Yaskawa INFORM job: DEMO_ROOF_SIDE_0625_3PAINT_44.JBI

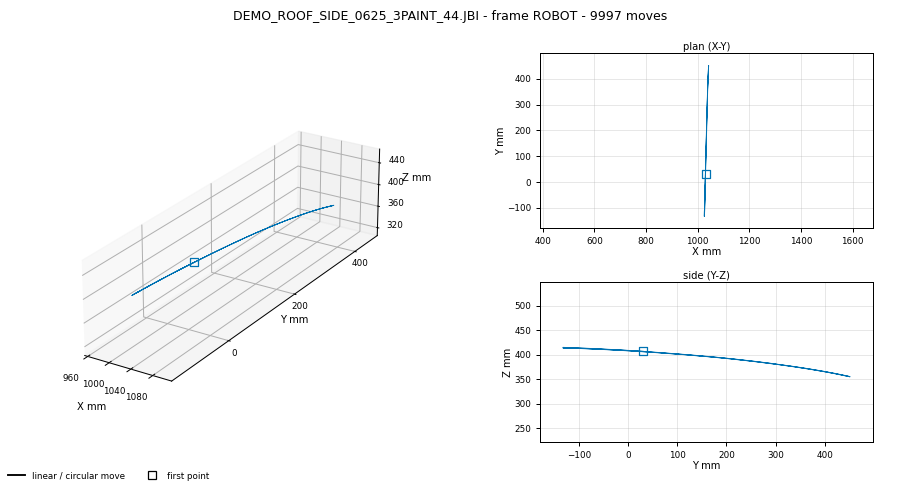
[picture p0: tool path of DEMO_ROOF_SIDE_0625_3PAINT_44.JBI in frame ROBOT, 9997 of 9997 moves have a stored position in this frame; points joined in program order, loops and branches not executed]
/JOB
//NAME DEMO_ROOF_SIDE_0625_3PAINT44
//POS
///NPOS 9997,0,0,0,0,0
///TOOL 0
///USER 0
///POSTYPE ROBOT
///RECTAN
///RCONF 1,0,0,0,0,0,0,0,0,0,0,0,0,0,0,0,0,0,0,0,0,0,0,0
C00000=1030.820,31.056,407.036,168.328,43.418,158.095
C00001=1030.814,30.807,407.052,168.325,43.419,158.095
C00002=1030.807,30.558,407.068,168.324,43.421,158.095
C00003=1030.801,30.309,407.084,168.321,43.422,158.095
C00004=1030.795,30.059,407.101,168.319,43.423,158.096
C00005=1030.788,29.809,407.116,168.316,43.425,158.096
C00006=1030.782,29.560,407.132,168.314,43.426,158.096
C00007=1030.776,29.310,407.148,168.312,43.427,158.096
C00008=1030.770,29.061,407.164,168.309,43.429,158.096
C00009=1030.764,28.812,407.180,168.306,43.431,158.096
C00010=1030.758,28.562,407.197,168.305,43.432,158.096
C00011=1030.750,28.276,407.215,168.302,43.433,158.096
C00012=1030.744,27.990,407.233,168.299,43.435,158.096
C00013=1030.737,27.704,407.251,168.297,43.437,158.096
C00014=1030.728,27.418,407.269,168.294,43.438,158.096
C00015=1030.722,27.169,407.286,168.291,43.440,158.096
C00016=1030.716,26.919,407.301,168.289,43.442,158.097
C00017=1030.710,26.670,407.317,168.287,43.443,158.097
C00018=1030.703,26.421,407.333,168.284,43.445,158.097
C00019=1030.697,26.171,407.349,168.281,43.446,158.097
C00020=1030.692,25.921,407.364,168.280,43.448,158.097
C00021=1030.685,25.672,407.380,168.277,43.449,158.097
C00022=1030.678,25.422,407.396,168.274,43.451,158.097
C00023=1030.672,25.173,407.412,168.272,43.452,158.097
C00024=1030.665,24.923,407.427,168.270,43.454,158.097
C00025=1030.660,24.674,407.444,168.267,43.456,158.097
C00026=1030.653,24.425,407.459,168.265,43.457,158.097
C00027=1030.647,24.175,407.475,168.263,43.459,158.098
C00028=1030.641,23.926,407.490,168.260,43.460,158.098
C00029=1030.635,23.677,407.507,168.257,43.462,158.098
C00030=1030.628,23.427,407.522,168.255,43.463,158.098
C00031=1030.622,23.178,407.538,168.253,43.464,158.098
C00032=1030.616,22.929,407.554,168.250,43.466,158.098
C00033=1030.610,22.679,407.569,168.248,43.467,158.098
C00034=1030.603,22.430,407.585,168.245,43.469,158.098
C00035=1030.597,22.181,407.600,168.243,43.470,158.098
C00036=1030.591,21.931,407.616,168.241,43.471,158.098
C00037=1030.584,21.682,407.632,168.238,43.473,158.098
C00038=1030.579,21.432,407.647,168.236,43.474,158.098
C00039=1030.572,21.183,407.663,168.234,43.476,158.098
C00040=1030.566,20.933,407.679,168.231,43.477,158.098
C00041=1030.560,20.684,407.694,168.228,43.479,158.099
C00042=1030.554,20.434,407.710,168.227,43.480,158.099
C00043=1030.547,20.185,407.725,168.224,43.482,158.099
C00044=1030.540,19.936,407.741,168.221,43.483,158.099
C00045=1030.535,19.686,407.756,168.220,43.485,158.099
C00046=1030.528,19.437,407.772,168.217,43.487,158.099
C00047=1030.523,19.187,407.788,168.214,43.488,158.099
C00048=1030.516,18.938,407.803,168.212,43.490,158.099
C00049=1030.509,18.688,407.818,168.210,43.491,158.099
C00050=1030.503,18.439,407.834,168.207,43.493,158.099
C00051=1030.497,18.189,407.849,168.204,43.494,158.099
C00052=1030.490,17.940,407.865,168.203,43.496,158.100
C00053=1030.484,17.690,407.880,168.200,43.498,158.100
C00054=1030.478,17.441,407.896,168.197,43.499,158.100
C00055=1030.472,17.191,407.911,168.195,43.500,158.100
C00056=1030.465,16.942,407.926,168.193,43.502,158.100
C00057=1030.459,16.692,407.942,168.190,43.504,158.100
C00058=1030.453,16.442,407.957,168.188,43.505,158.100
C00059=1030.446,16.193,407.973,168.186,43.506,158.100
C00060=1030.440,15.944,407.988,168.183,43.508,158.100
C00061=1030.434,15.694,408.004,168.180,43.509,158.100
C00062=1030.428,15.445,408.019,168.178,43.511,158.100
C00063=1030.421,15.195,408.034,168.176,43.512,158.100
C00064=1030.416,14.947,408.050,168.173,43.514,158.101
C00065=1030.409,14.697,408.065,168.171,43.515,158.101
C00066=1030.403,14.447,408.080,168.169,43.517,158.101
C00067=1030.396,14.198,408.096,168.166,43.518,158.101
C00068=1030.391,13.948,408.111,168.164,43.520,158.101
C00069=1030.384,13.699,408.126,168.161,43.521,158.101
C00070=1030.378,13.449,408.142,168.159,43.523,158.101
C00071=1030.371,13.200,408.157,168.156,43.525,158.101
C00072=1030.365,12.950,408.172,168.154,43.526,158.101
C00073=1030.359,12.701,408.187,168.151,43.528,158.101
C00074=1030.352,12.451,408.202,168.149,43.530,158.101
C00075=1030.345,12.166,408.219,168.146,43.531,158.101
C00076=1030.338,11.882,408.236,168.143,43.533,158.102
C00077=1030.330,11.597,408.253,168.141,43.535,158.102
C00078=1030.323,11.312,408.271,168.137,43.537,158.102
C00079=1030.317,11.063,408.285,168.136,43.538,158.102
C00080=1030.310,10.813,408.300,168.133,43.540,158.102
C00081=1030.304,10.563,408.315,168.130,43.541,158.102
C00082=1030.298,10.314,408.330,168.127,43.543,158.102
C00083=1030.291,10.065,408.346,168.126,43.544,158.102
C00084=1030.285,9.816,408.361,168.123,43.546,158.102
C00085=1030.279,9.566,408.376,168.120,43.548,158.103
C00086=1030.272,9.317,408.390,168.117,43.549,158.102
C00087=1030.266,9.067,408.405,168.116,43.551,158.103
C00088=1030.260,8.817,408.420,168.113,43.553,158.103
C00089=1030.253,8.568,408.435,168.110,43.554,158.103
C00090=1030.247,8.319,408.450,168.108,43.556,158.103
C00091=1030.241,8.069,408.465,168.105,43.558,158.103
C00092=1030.234,7.820,408.480,168.103,43.559,158.103
C00093=1030.228,7.570,408.495,168.101,43.561,158.103
C00094=1030.222,7.321,408.510,168.098,43.562,158.103
C00095=1030.215,7.071,408.525,168.095,43.564,158.103
C00096=1030.209,6.822,408.540,168.094,43.566,158.104
C00097=1030.203,6.572,408.555,168.091,43.567,158.104
C00098=1030.197,6.323,408.570,168.088,43.569,158.104
C00099=1030.190,6.073,408.585,168.085,43.570,158.104
C00100=1030.184,5.824,408.599,168.084,43.572,158.104
C00101=1030.178,5.574,408.614,168.081,43.573,158.104
C00102=1030.172,5.325,408.629,168.078,43.575,158.104
C00103=1030.165,5.075,408.644,168.076,43.576,158.104
C00104=1030.159,4.825,408.659,168.074,43.577,158.104
C00105=1030.153,4.576,408.674,168.071,43.579,158.104
C00106=1030.147,4.327,408.689,168.068,43.581,158.104
C00107=1030.140,4.077,408.704,168.066,43.582,158.104
C00108=1030.134,3.827,408.719,168.063,43.584,158.104
C00109=1030.128,3.579,408.733,168.061,43.585,158.104
C00110=1030.122,3.329,408.748,168.059,43.587,158.105
C00111=1030.115,3.079,408.763,168.056,43.588,158.105
C00112=1030.110,2.830,408.778,168.053,43.590,158.105
C00113=1030.103,2.581,408.793,168.051,43.592,158.105
C00114=1030.097,2.331,408.807,168.049,43.593,158.105
C00115=1030.090,2.081,408.822,168.046,43.595,158.105
C00116=1030.085,1.832,408.836,168.043,43.596,158.105
C00117=1030.079,1.582,408.851,168.042,43.598,158.105
C00118=1030.072,1.332,408.866,168.039,43.599,158.105
C00119=1030.066,1.083,408.881,168.036,43.601,158.105
C00120=1030.060,0.834,408.896,168.033,43.602,158.105
C00121=1030.054,0.584,408.911,168.032,43.604,158.105
C00122=1030.048,0.335,408.925,168.029,43.605,158.105
C00123=1030.042,0.086,408.940,168.026,43.607,158.106
C00124=1030.035,-0.165,408.954,168.023,43.608,158.106
C00125=1030.030,-0.414,408.969,168.021,43.610,158.106
C00126=1030.023,-0.663,408.983,168.019,43.612,158.106
C00127=1030.016,-0.913,408.998,168.016,43.613,158.106
C00128=1030.010,-1.162,409.013,168.014,43.615,158.106
C00129=1030.004,-1.411,409.028,168.011,43.616,158.106
C00130=1029.999,-1.661,409.042,168.009,43.618,158.106
C00131=1029.992,-1.911,409.057,168.006,43.619,158.106
C00132=1029.986,-2.160,409.072,168.004,43.621,158.106
C00133=1029.980,-2.409,409.086,168.001,43.622,158.106
C00134=1029.974,-2.659,409.101,167.999,43.624,158.106
C00135=1029.968,-2.908,409.115,167.996,43.625,158.106
C00136=1029.962,-3.158,409.130,167.994,43.627,158.107
C00137=1029.955,-3.408,409.145,167.991,43.628,158.107
C00138=1029.950,-3.657,409.159,167.989,43.630,158.107
C00139=1029.942,-3.940,409.176,167.985,43.631,158.107
C00140=1029.935,-4.223,409.191,167.983,43.633,158.107
C00141=1029.928,-4.505,409.208,167.980,43.635,158.107
C00142=1029.921,-4.789,409.225,167.978,43.637,158.107
C00143=1029.915,-5.038,409.238,167.975,43.639,158.107
C00144=1029.908,-5.288,409.253,167.972,43.641,158.107
C00145=1029.902,-5.537,409.267,167.969,43.642,158.107
C00146=1029.896,-5.787,409.281,167.967,43.644,158.107
C00147=1029.889,-6.036,409.296,167.964,43.646,158.107
C00148=1029.883,-6.286,409.309,167.962,43.647,158.108
C00149=1029.877,-6.535,409.324,167.960,43.649,158.108
C00150=1029.871,-6.784,409.339,167.957,43.650,158.108
C00151=1029.864,-7.034,409.352,167.954,43.652,158.108
C00152=1029.858,-7.284,409.367,167.952,43.654,158.108
C00153=1029.851,-7.533,409.381,167.949,43.655,158.108
C00154=1029.845,-7.783,409.396,167.946,43.657,158.108
C00155=1029.840,-8.032,409.409,167.945,43.658,158.108
C00156=1029.832,-8.282,409.424,167.942,43.660,158.108
C00157=1029.827,-8.531,409.438,167.939,43.661,158.108
C00158=1029.820,-8.781,409.452,167.936,43.663,158.108
C00159=1029.814,-9.030,409.466,167.934,43.665,158.109
C00160=1029.808,-9.280,409.481,167.931,43.666,158.109
C00161=1029.801,-9.530,409.494,167.928,43.668,158.109
C00162=1029.795,-9.779,409.509,167.927,43.670,158.109
C00163=1029.789,-10.029,409.523,167.924,43.671,158.109
C00164=1029.783,-10.278,409.537,167.921,43.673,158.109
C00165=1029.776,-10.528,409.551,167.919,43.675,158.109
C00166=1029.770,-10.777,409.565,167.916,43.676,158.109
C00167=1029.764,-11.027,409.580,167.913,43.678,158.109
C00168=1029.758,-11.276,409.593,167.911,43.680,158.109
C00169=1029.752,-11.526,409.608,167.909,43.681,158.109
C00170=1029.745,-11.775,409.621,167.906,43.683,158.109
C00171=1029.740,-12.025,409.635,167.903,43.684,158.109
C00172=1029.733,-12.274,409.649,167.901,43.686,158.110
C00173=1029.727,-12.524,409.663,167.898,43.688,158.110
C00174=1029.721,-12.773,409.678,167.895,43.689,158.110
C00175=1029.715,-13.023,409.691,167.893,43.691,158.110
C00176=1029.709,-13.273,409.706,167.891,43.693,158.110
C00177=1029.702,-13.521,409.720,167.888,43.694,158.110
C00178=1029.696,-13.772,409.734,167.885,43.696,158.110
C00179=1029.690,-14.021,409.747,167.883,43.697,158.110
C00180=1029.684,-14.270,409.762,167.880,43.699,158.110
C00181=1029.678,-14.520,409.776,167.877,43.701,158.110
C00182=1029.672,-14.770,409.789,167.875,43.702,158.110
C00183=1029.666,-15.020,409.803,167.873,43.704,158.110
C00184=1029.659,-15.268,409.817,167.870,43.705,158.110
C00185=1029.653,-15.519,409.832,167.867,43.707,158.111
C00186=1029.647,-15.768,409.845,167.865,43.709,158.111
C00187=1029.640,-16.018,409.859,167.862,43.710,158.111
C00188=1029.634,-16.267,409.873,167.859,43.712,158.111
C00189=1029.628,-16.516,409.886,167.857,43.714,158.111
C00190=1029.621,-16.766,409.900,167.854,43.716,158.111
C00191=1029.616,-17.016,409.914,167.851,43.717,158.111
C00192=1029.609,-17.266,409.928,167.849,43.719,158.111
C00193=1029.603,-17.515,409.941,167.847,43.720,158.111
C00194=1029.597,-17.764,409.955,167.844,43.722,158.111
C00195=1029.590,-18.014,409.969,167.842,43.723,158.111
C00196=1029.584,-18.263,409.982,167.839,43.725,158.112
C00197=1029.578,-18.513,409.997,167.836,43.727,158.112
C00198=1029.572,-18.763,410.010,167.834,43.729,158.112
C00199=1029.565,-19.012,410.023,167.831,43.730,158.112
C00200=1029.559,-19.262,410.037,167.828,43.732,158.112
C00201=1029.553,-19.511,410.051,167.826,43.734,158.112
C00202=1029.547,-19.761,410.064,167.823,43.736,158.112
C00203=1029.540,-20.042,410.080,167.820,43.738,158.112
C00204=1029.533,-20.323,410.095,167.817,43.739,158.112
C00205=1029.525,-20.605,410.110,167.814,43.741,158.112
C00206=1029.518,-20.886,410.126,167.811,43.743,158.112
C00207=1029.512,-21.135,410.139,167.809,43.745,158.113
C00208=1029.506,-21.385,410.153,167.806,43.747,158.113
C00209=1029.500,-21.635,410.167,167.803,43.748,158.113
C00210=1029.493,-21.884,410.180,167.800,43.750,158.113
C00211=1029.487,-22.134,410.193,167.798,43.752,158.113
C00212=1029.482,-22.383,410.207,167.795,43.754,158.113
C00213=1029.475,-22.633,410.221,167.793,43.755,158.113
C00214=1029.469,-22.882,410.234,167.791,43.757,158.113
C00215=1029.463,-23.132,410.248,167.788,43.759,158.113
C00216=1029.456,-23.382,410.261,167.785,43.760,158.113
C00217=1029.450,-23.631,410.275,167.783,43.762,158.113
C00218=1029.444,-23.880,410.288,167.780,43.764,158.113
C00219=1029.438,-24.130,410.302,167.777,43.765,158.113
C00220=1029.432,-24.380,410.316,167.775,43.767,158.114
C00221=1029.425,-24.629,410.329,167.772,43.769,158.114
C00222=1029.419,-24.878,410.342,167.769,43.770,158.114
C00223=1029.414,-25.128,410.356,167.766,43.772,158.114
C00224=1029.407,-25.378,410.370,167.764,43.774,158.114
C00225=1029.401,-25.628,410.382,167.761,43.775,158.114
C00226=1029.395,-25.877,410.395,167.758,43.777,158.114
C00227=1029.389,-26.127,410.409,167.756,43.779,158.114
C00228=1029.383,-26.376,410.423,167.754,43.780,158.114
C00229=1029.376,-26.626,410.436,167.751,43.782,158.114
C00230=1029.370,-26.875,410.449,167.749,43.783,158.114
C00231=1029.365,-27.125,410.463,167.746,43.785,158.114
C00232=1029.359,-27.375,410.476,167.743,43.787,158.115
C00233=1029.352,-27.625,410.489,167.741,43.788,158.115
C00234=1029.346,-27.874,410.503,167.738,43.790,158.115
C00235=1029.339,-28.123,410.516,167.735,43.792,158.115
C00236=1029.334,-28.373,410.529,167.732,43.793,158.115
C00237=1029.327,-28.622,410.542,167.730,43.795,158.115
C00238=1029.321,-28.872,410.555,167.727,43.797,158.115
C00239=1029.314,-29.122,410.569,167.725,43.799,158.115
C00240=1029.308,-29.371,410.581,167.722,43.801,158.115
C00241=1029.302,-29.621,410.595,167.719,43.802,158.115
C00242=1029.296,-29.870,410.608,167.716,43.804,158.115
C00243=1029.289,-30.121,410.621,167.714,43.806,158.116
C00244=1029.283,-30.370,410.634,167.711,43.808,158.116
C00245=1029.277,-30.619,410.647,167.709,43.810,158.116
C00246=1029.271,-30.869,410.660,167.706,43.811,158.116
C00247=1029.265,-31.118,410.673,167.703,43.813,158.116
C00248=1029.259,-31.367,410.686,167.701,43.815,158.116
C00249=1029.253,-31.617,410.699,167.698,43.817,158.116
C00250=1029.246,-31.867,410.713,167.695,43.818,158.116
C00251=1029.240,-32.117,410.726,167.692,43.820,158.116
C00252=1029.234,-32.366,410.738,167.690,43.822,158.116
C00253=1029.228,-32.616,410.752,167.687,43.824,158.116
C00254=1029.222,-32.866,410.764,167.685,43.826,158.117
C00255=1029.216,-33.115,410.777,167.682,43.827,158.117
C00256=1029.209,-33.364,410.791,167.679,43.829,158.117
C00257=1029.203,-33.614,410.803,167.676,43.831,158.117
C00258=1029.196,-33.864,410.816,167.674,43.833,158.117
C00259=1029.190,-34.114,410.829,167.671,43.834,158.117
C00260=1029.184,-34.363,410.842,167.668,43.836,158.117
C00261=1029.178,-34.613,410.855,167.666,43.838,158.117
C00262=1029.172,-34.862,410.868,167.663,43.840,158.117
C00263=1029.166,-35.112,410.881,167.660,43.841,158.117
C00264=1029.159,-35.361,410.894,167.658,43.843,158.117
C00265=1029.154,-35.611,410.906,167.655,43.845,158.117
C00266=1029.147,-35.860,410.920,167.652,43.846,158.118
C00267=1029.141,-36.141,410.934,167.649,43.849,158.118
C00268=1029.134,-36.421,410.948,167.646,43.850,158.118
C00269=1029.127,-36.702,410.963,167.643,43.852,158.118
C00270=1029.120,-36.982,410.977,167.640,43.854,158.118
C00271=1029.114,-37.232,410.990,167.637,43.856,158.118
C00272=1029.108,-37.481,411.003,167.634,43.858,158.118
C00273=1029.102,-37.731,411.016,167.632,43.859,158.118
C00274=1029.095,-37.980,411.029,167.629,43.861,158.118
C00275=1029.090,-38.230,411.042,167.626,43.863,158.118
C00276=1029.084,-38.480,411.054,167.624,43.864,158.118
C00277=1029.077,-38.729,411.067,167.621,43.866,158.118
C00278=1029.072,-38.979,411.080,167.618,43.868,158.118
C00279=1029.065,-39.228,411.093,167.616,43.870,158.119
C00280=1029.059,-39.478,411.105,167.613,43.871,158.119
C00281=1029.053,-39.728,411.118,167.610,43.873,158.119
C00282=1029.047,-39.978,411.130,167.608,43.875,158.119
C00283=1029.040,-40.227,411.143,167.605,43.877,158.119
C00284=1029.034,-40.476,411.155,167.602,43.879,158.119
C00285=1029.028,-40.726,411.168,167.600,43.881,158.119
C00286=1029.022,-40.976,411.181,167.596,43.882,158.119
C00287=1029.015,-41.225,411.193,167.593,43.884,158.119
C00288=1029.009,-41.475,411.206,167.591,43.886,158.119
C00289=1029.003,-41.725,411.218,167.588,43.888,158.119
C00290=1028.996,-41.974,411.231,167.585,43.890,158.120
C00291=1028.991,-42.224,411.244,167.583,43.892,158.120
C00292=1028.985,-42.474,411.256,167.580,43.894,158.120
C00293=1028.978,-42.723,411.268,167.578,43.896,158.120
C00294=1028.972,-42.973,411.281,167.575,43.897,158.120
C00295=1028.966,-43.222,411.294,167.572,43.899,158.120
C00296=1028.959,-43.472,411.306,167.569,43.901,158.120
C00297=1028.953,-43.722,411.318,167.567,43.903,158.120
C00298=1028.948,-43.971,411.331,167.563,43.905,158.120
C00299=1028.941,-44.221,411.343,167.561,43.907,158.120
C00300=1028.935,-44.471,411.355,167.558,43.909,158.121
C00301=1028.929,-44.720,411.368,167.555,43.910,158.120
C00302=1028.923,-44.969,411.380,167.552,43.912,158.121
C00303=1028.917,-45.219,411.393,167.550,43.914,158.121
C00304=1028.911,-45.469,411.405,167.547,43.916,158.121
C00305=1028.904,-45.719,411.417,167.545,43.917,158.121
C00306=1028.898,-45.969,411.430,167.542,43.919,158.121
C00307=1028.893,-46.218,411.442,167.539,43.921,158.121
C00308=1028.886,-46.467,411.454,167.536,43.923,158.121
C00309=1028.880,-46.717,411.467,167.534,43.924,158.121
C00310=1028.874,-46.966,411.480,167.531,43.926,158.121
C00311=1028.867,-47.216,411.492,167.528,43.928,158.121
C00312=1028.862,-47.466,411.504,167.525,43.930,158.122
C00313=1028.856,-47.715,411.517,167.522,43.932,158.122
C00314=1028.850,-47.965,411.529,167.520,43.933,158.122
C00315=1028.844,-48.215,411.541,167.517,43.935,158.122
C00316=1028.838,-48.464,411.554,167.514,43.937,158.122
C00317=1028.831,-48.714,411.566,167.512,43.939,158.122
C00318=1028.826,-48.963,411.578,167.509,43.940,158.122
C00319=1028.819,-49.213,411.590,167.506,43.942,158.122
C00320=1028.813,-49.463,411.602,167.504,43.944,158.122
C00321=1028.807,-49.713,411.615,167.501,43.946,158.122
C00322=1028.801,-49.962,411.627,167.498,43.948,158.122
C00323=1028.795,-50.211,411.639,167.494,43.950,158.122
C00324=1028.790,-50.461,411.652,167.492,43.951,158.122
C00325=1028.783,-50.711,411.664,167.489,43.953,158.123
C00326=1028.777,-50.961,411.675,167.487,43.955,158.123
C00327=1028.771,-51.211,411.687,167.484,43.957,158.123
C00328=1028.765,-51.460,411.699,167.481,43.959,158.123
C00329=1028.758,-51.709,411.711,167.479,43.961,158.123
C00330=1028.752,-51.959,411.724,167.475,43.963,158.123
C00331=1028.743,-52.314,411.740,167.472,43.966,158.123
C00332=1028.734,-52.667,411.757,167.467,43.969,158.123
C00333=1028.725,-53.021,411.774,167.464,43.972,158.124
C00334=1028.717,-53.376,411.791,167.459,43.975,158.124
C00335=1028.710,-53.625,411.803,167.457,43.977,158.124
C00336=1028.704,-53.874,411.814,167.454,43.978,158.124
C00337=1028.698,-54.124,411.825,167.451,43.980,158.124
C00338=1028.692,-54.374,411.838,167.449,43.982,158.124
C00339=1028.685,-54.624,411.850,167.445,43.984,158.124
C00340=1028.679,-54.873,411.861,167.443,43.986,158.124
C00341=1028.673,-55.123,411.873,167.440,43.988,158.124
C00342=1028.667,-55.373,411.885,167.437,43.990,158.125
C00343=1028.661,-55.622,411.897,167.435,43.992,158.125
C00344=1028.654,-55.872,411.908,167.431,43.994,158.125
C00345=1028.648,-56.121,411.920,167.428,43.996,158.125
C00346=1028.642,-56.371,411.932,167.426,43.998,158.125
C00347=1028.636,-56.621,411.943,167.423,44.000,158.125
C00348=1028.629,-56.870,411.955,167.421,44.002,158.125
C00349=1028.623,-57.120,411.967,167.417,44.004,158.125
C00350=1028.618,-57.370,411.979,167.414,44.006,158.125
C00351=1028.611,-57.619,411.991,167.412,44.008,158.125
C00352=1028.605,-57.869,412.002,167.409,44.010,158.126
C00353=1028.599,-58.118,412.014,167.406,44.012,158.126
C00354=1028.593,-58.369,412.026,167.404,44.014,158.126
C00355=1028.587,-58.618,412.037,167.400,44.016,158.126
C00356=1028.580,-58.867,412.049,167.397,44.018,158.126
C00357=1028.574,-59.117,412.060,167.395,44.019,158.126
C00358=1028.568,-59.366,412.072,167.392,44.021,158.126
C00359=1028.562,-59.617,412.084,167.390,44.023,158.126
C00360=1028.556,-59.866,412.096,167.386,44.025,158.126
C00361=1028.550,-60.116,412.107,167.383,44.027,158.126
C00362=1028.543,-60.365,412.119,167.381,44.029,158.126
C00363=1028.538,-60.615,412.130,167.378,44.031,158.127
C00364=1028.532,-60.865,412.142,167.375,44.033,158.127
C00365=1028.526,-61.114,412.153,167.372,44.035,158.127
C00366=1028.519,-61.364,412.165,167.369,44.037,158.127
C00367=1028.513,-61.614,412.176,167.367,44.039,158.127
C00368=1028.508,-61.863,412.188,167.364,44.041,158.127
C00369=1028.501,-62.113,412.199,167.361,44.043,158.127
C00370=1028.495,-62.362,412.211,167.358,44.045,158.127
C00371=1028.489,-62.613,412.222,167.355,44.047,158.127
C00372=1028.483,-62.861,412.234,167.352,44.049,158.127
C00373=1028.477,-63.112,412.246,167.350,44.051,158.128
C00374=1028.471,-63.361,412.257,167.347,44.053,158.128
C00375=1028.465,-63.611,412.269,167.344,44.055,158.128
C00376=1028.459,-63.860,412.279,167.341,44.057,158.128
C00377=1028.453,-64.110,412.291,167.338,44.059,158.128
C00378=1028.448,-64.360,412.303,167.336,44.061,158.128
C00379=1028.441,-64.609,412.315,167.333,44.063,158.128
C00380=1028.435,-64.859,412.326,167.330,44.064,158.128
C00381=1028.429,-65.109,412.337,167.327,44.067,158.128
C00382=1028.423,-65.358,412.349,167.324,44.068,158.128
C00383=1028.417,-65.608,412.360,167.322,44.070,158.129
C00384=1028.412,-65.858,412.371,167.319,44.072,158.129
C00385=1028.405,-66.107,412.383,167.316,44.074,158.129
C00386=1028.399,-66.357,412.394,167.313,44.076,158.129
C00387=1028.393,-66.570,412.404,167.311,44.077,158.129
C00388=1028.389,-66.783,412.414,167.308,44.079,158.129
C00389=1028.384,-66.997,412.423,167.306,44.081,158.129
C00390=1028.379,-67.209,412.433,167.303,44.083,158.129
C00391=1028.373,-67.423,412.443,167.301,44.084,158.129
C00392=1028.368,-67.636,412.453,167.299,44.086,158.129
C00393=1028.364,-67.849,412.462,167.296,44.087,158.129
C00394=1028.358,-68.062,412.472,167.294,44.089,158.129
C00395=1028.352,-68.344,412.484,167.290,44.091,158.129
C00396=1028.345,-68.626,412.498,167.287,44.093,158.130
C00397=1028.338,-68.908,412.510,167.284,44.096,158.130
C00398=1028.331,-69.191,412.523,167.281,44.098,158.130
C00399=1028.325,-69.440,412.534,167.278,44.100,158.130
C00400=1028.320,-69.690,412.545,167.275,44.102,158.130
C00401=1028.314,-69.940,412.557,167.272,44.104,158.130
C00402=1028.308,-70.189,412.568,167.269,44.106,158.130
C00403=1028.302,-70.439,412.579,167.266,44.107,158.130
C00404=1028.296,-70.689,412.590,167.264,44.109,158.130
C00405=1028.290,-70.938,412.601,167.261,44.111,158.130
C00406=1028.284,-71.188,412.612,167.257,44.113,158.130
C00407=1028.278,-71.437,412.624,167.255,44.115,158.130
C00408=1028.273,-71.687,412.635,167.252,44.117,158.131
C00409=1028.267,-71.937,412.646,167.250,44.119,158.131
C00410=1028.261,-72.187,412.658,167.247,44.121,158.131
C00411=1028.255,-72.436,412.668,167.243,44.123,158.131
C00412=1028.249,-72.686,412.679,167.241,44.125,158.131
C00413=1028.243,-72.936,412.691,167.238,44.127,158.131
C00414=1028.237,-73.185,412.701,167.235,44.129,158.131
C00415=1028.232,-73.435,412.713,167.233,44.131,158.131
C00416=1028.225,-73.685,412.725,167.229,44.132,158.131
C00417=1028.220,-73.934,412.736,167.226,44.134,158.131
C00418=1028.214,-74.184,412.747,167.224,44.136,158.131
C00419=1028.208,-74.433,412.757,167.221,44.138,158.131
C00420=1028.202,-74.684,412.769,167.219,44.140,158.132
C00421=1028.196,-74.933,412.780,167.215,44.143,158.132
C00422=1028.190,-75.182,412.790,167.212,44.145,158.132
C00423=1028.184,-75.433,412.800,167.210,44.147,158.132
C00424=1028.178,-75.682,412.811,167.206,44.149,158.132
C00425=1028.172,-75.932,412.822,167.204,44.151,158.132
C00426=1028.166,-76.181,412.833,167.201,44.153,158.132
C00427=1028.160,-76.432,412.844,167.198,44.155,158.132
C00428=1028.154,-76.681,412.855,167.195,44.157,158.132
C00429=1028.148,-76.930,412.865,167.192,44.159,158.132
C00430=1028.141,-77.181,412.877,167.189,44.161,158.133
C00431=1028.136,-77.430,412.888,167.187,44.163,158.133
C00432=1028.130,-77.679,412.898,167.183,44.165,158.133
C00433=1028.125,-77.930,412.909,167.181,44.167,158.133
C00434=1028.119,-78.179,412.920,167.178,44.169,158.133
C00435=1028.112,-78.429,412.930,167.175,44.171,158.133
C00436=1028.106,-78.678,412.941,167.172,44.173,158.133
C00437=1028.100,-78.928,412.952,167.169,44.175,158.133
C00438=1028.094,-79.177,412.963,167.167,44.177,158.133
C00439=1028.088,-79.428,412.973,167.163,44.179,158.133
C00440=1028.083,-79.678,412.984,167.160,44.181,158.134
C00441=1028.076,-79.927,412.994,167.158,44.183,158.134
C00442=1028.070,-80.176,413.005,167.154,44.186,158.134
C00443=1028.065,-80.427,413.016,167.152,44.188,158.134
C00444=1028.058,-80.676,413.026,167.149,44.190,158.134
C00445=1028.052,-80.926,413.037,167.145,44.192,158.134
C00446=1028.046,-81.176,413.047,167.143,44.195,158.134
C00447=1028.040,-81.425,413.057,167.140,44.196,158.134
C00448=1028.035,-81.675,413.068,167.137,44.199,158.135
C00449=1028.028,-81.925,413.078,167.134,44.201,158.135
C00450=1028.022,-82.175,413.089,167.132,44.203,158.135
C00451=1028.016,-82.424,413.099,167.128,44.205,158.135
C00452=1028.010,-82.674,413.110,167.126,44.207,158.135
C00453=1028.004,-82.923,413.120,167.123,44.210,158.135
C00454=1027.998,-83.173,413.130,167.119,44.212,158.135
C00455=1027.992,-83.423,413.141,167.117,44.214,158.135
C00456=1027.985,-83.673,413.152,167.114,44.216,158.135
C00457=1027.980,-83.923,413.162,167.111,44.219,158.136
C00458=1027.974,-84.172,413.172,167.108,44.221,158.136
C00459=1027.967,-84.457,413.184,167.105,44.223,158.136
C00460=1027.961,-84.740,413.196,167.101,44.226,158.136
C00461=1027.953,-85.025,413.207,167.099,44.228,158.136
C00462=1027.946,-85.309,413.219,167.095,44.230,158.136
C00463=1027.941,-85.559,413.230,167.091,44.232,158.136
C00464=1027.935,-85.809,413.239,167.089,44.234,158.136
C00465=1027.929,-86.058,413.250,167.086,44.237,158.137
C00466=1027.923,-86.308,413.260,167.083,44.239,158.137
C00467=1027.917,-86.557,413.271,167.080,44.241,158.137
C00468=1027.911,-86.807,413.280,167.078,44.243,158.137
C00469=1027.905,-87.057,413.291,167.074,44.246,158.137
C00470=1027.900,-87.307,413.301,167.071,44.248,158.137
C00471=1027.893,-87.556,413.311,167.069,44.250,158.137
C00472=1027.888,-87.806,413.322,167.065,44.252,158.137
C00473=1027.881,-88.055,413.332,167.063,44.255,158.138
C00474=1027.876,-88.305,413.342,167.060,44.256,158.138
C00475=1027.870,-88.555,413.352,167.057,44.259,158.138
C00476=1027.864,-88.805,413.363,167.054,44.261,158.138
C00477=1027.858,-89.055,413.372,167.052,44.263,158.138
C00478=1027.852,-89.304,413.383,167.048,44.265,158.138
C00479=1027.846,-89.554,413.393,167.045,44.267,158.138
C00480=1027.840,-89.804,413.403,167.043,44.269,158.138
C00481=1027.834,-90.053,413.413,167.039,44.271,158.138
C00482=1027.828,-90.303,413.423,167.037,44.274,158.139
C00483=1027.822,-90.553,413.433,167.034,44.276,158.139
C00484=1027.817,-90.803,413.444,167.030,44.278,158.139
C00485=1027.810,-91.052,413.453,167.028,44.280,158.139
C00486=1027.805,-91.302,413.463,167.025,44.283,158.139
C00487=1027.798,-91.552,413.474,167.022,44.285,158.139
C00488=1027.793,-91.802,413.484,167.019,44.287,158.139
C00489=1027.787,-92.052,413.493,167.016,44.289,158.139
C00490=1027.781,-92.301,413.504,167.013,44.291,158.139
C00491=1027.775,-92.551,413.514,167.010,44.293,158.140
C00492=1027.769,-92.801,413.524,167.008,44.295,158.140
C00493=1027.763,-93.050,413.534,167.004,44.298,158.140
C00494=1027.758,-93.300,413.544,167.002,44.299,158.140
C00495=1027.751,-93.550,413.554,166.999,44.301,158.140
C00496=1027.747,-93.799,413.564,166.996,44.304,158.140
C00497=1027.740,-94.049,413.574,166.993,44.306,158.140
C00498=1027.735,-94.299,413.584,166.989,44.308,158.140
C00499=1027.728,-94.548,413.594,166.987,44.310,158.140
C00500=1027.723,-94.799,413.604,166.984,44.313,158.140
C00501=1027.717,-95.048,413.613,166.981,44.315,158.141
C00502=1027.711,-95.298,413.624,166.978,44.317,158.141
C00503=1027.705,-95.548,413.634,166.975,44.319,158.141
C00504=1027.700,-95.797,413.644,166.972,44.321,158.141
C00505=1027.694,-96.047,413.653,166.969,44.324,158.141
C00506=1027.689,-96.297,413.663,166.967,44.326,158.141
C00507=1027.682,-96.547,413.673,166.963,44.328,158.141
C00508=1027.677,-96.796,413.684,166.960,44.330,158.141
C00509=1027.671,-97.045,413.693,166.958,44.332,158.141
C00510=1027.666,-97.295,413.703,166.954,44.335,158.141
C00511=1027.659,-97.545,413.713,166.952,44.337,158.142
C00512=1027.654,-97.795,413.723,166.949,44.338,158.142
C00513=1027.648,-98.045,413.733,166.946,44.341,158.142
C00514=1027.642,-98.295,413.742,166.943,44.343,158.142
C00515=1027.636,-98.544,413.751,166.939,44.345,158.142
C00516=1027.630,-98.794,413.761,166.937,44.348,158.142
C00517=1027.624,-99.044,413.771,166.934,44.350,158.142
C00518=1027.618,-99.294,413.781,166.931,44.352,158.142
C00519=1027.612,-99.544,413.790,166.928,44.355,158.143
C00520=1027.607,-99.793,413.799,166.925,44.357,158.143
C00521=1027.601,-100.043,413.810,166.922,44.360,158.143
C00522=1027.595,-100.293,413.819,166.920,44.362,158.143
C00523=1027.588,-100.579,413.830,166.916,44.364,158.143
C00524=1027.582,-100.866,413.841,166.913,44.366,158.143
C00525=1027.575,-101.152,413.852,166.909,44.369,158.143
C00526=1027.568,-101.439,413.863,166.906,44.372,158.144
C00527=1027.563,-101.688,413.872,166.903,44.374,158.144
C00528=1027.556,-101.938,413.881,166.900,44.377,158.144
C00529=1027.550,-102.188,413.891,166.897,44.379,158.144
C00530=1027.545,-102.438,413.901,166.894,44.381,158.144
C00531=1027.539,-102.687,413.910,166.891,44.384,158.144
C00532=1027.533,-102.937,413.920,166.889,44.386,158.144
C00533=1027.527,-103.187,413.929,166.885,44.388,158.144
C00534=1027.522,-103.436,413.938,166.883,44.390,158.144
C00535=1027.515,-103.686,413.947,166.879,44.393,158.145
C00536=1027.510,-103.936,413.958,166.877,44.395,158.145
C00537=1027.504,-104.185,413.967,166.874,44.397,158.145
C00538=1027.498,-104.435,413.976,166.870,44.399,158.145
C00539=1027.492,-104.685,413.985,166.868,44.402,158.145
C00540=1027.487,-104.935,413.994,166.864,44.404,158.145
C00541=1027.481,-105.184,414.004,166.862,44.407,158.145
C00542=1027.475,-105.434,414.014,166.859,44.409,158.145
C00543=1027.470,-105.684,414.023,166.856,44.411,158.146
C00544=1027.464,-105.934,414.032,166.853,44.414,158.146
C00545=1027.458,-106.184,414.042,166.850,44.416,158.146
C00546=1027.452,-106.433,414.051,166.847,44.418,158.146
C00547=1027.446,-106.683,414.060,166.844,44.421,158.146
C00548=1027.440,-106.933,414.069,166.841,44.422,158.146
C00549=1027.434,-107.182,414.079,166.838,44.425,158.146
C00550=1027.429,-107.433,414.088,166.835,44.427,158.146
C00551=1027.423,-107.683,414.098,166.832,44.430,158.147
C00552=1027.418,-107.932,414.107,166.829,44.432,158.147
C00553=1027.412,-108.182,414.116,166.826,44.435,158.147
C00554=1027.406,-108.431,414.125,166.823,44.437,158.147
C00555=1027.400,-108.681,414.134,166.820,44.440,158.147
C00556=1027.394,-108.932,414.143,166.818,44.442,158.147
C00557=1027.389,-109.181,414.152,166.814,44.444,158.147
C00558=1027.383,-109.431,414.161,166.812,44.446,158.147
C00559=1027.377,-109.680,414.171,166.808,44.449,158.148
C00560=1027.371,-109.930,414.180,166.806,44.451,158.148
C00561=1027.365,-110.179,414.188,166.802,44.454,158.148
C00562=1027.359,-110.429,414.198,166.800,44.456,158.148
C00563=1027.353,-110.680,414.206,166.796,44.459,158.148
C00564=1027.347,-110.929,414.216,166.794,44.461,158.148
C00565=1027.341,-111.179,414.224,166.791,44.463,158.149
C00566=1027.336,-111.428,414.234,166.788,44.466,158.149
C00567=1027.330,-111.679,414.243,166.785,44.468,158.149
C00568=1027.324,-111.928,414.252,166.782,44.470,158.149
C00569=1027.319,-112.178,414.261,166.779,44.473,158.149
C00570=1027.313,-112.427,414.270,166.776,44.475,158.149
C00571=1027.307,-112.678,414.279,166.773,44.478,158.149
C00572=1027.302,-112.927,414.288,166.770,44.480,158.149
C00573=1027.296,-113.177,414.297,166.767,44.482,158.149
C00574=1027.290,-113.426,414.306,166.765,44.485,158.150
C00575=1027.284,-113.677,414.315,166.761,44.487,158.150
C00576=1027.279,-113.926,414.323,166.758,44.489,158.150
C00577=1027.273,-114.176,414.333,166.755,44.492,158.150
C00578=1027.268,-114.426,414.341,166.752,44.494,158.150
C00579=1027.261,-114.676,414.351,166.749,44.496,158.150
C00580=1027.256,-114.925,414.359,166.746,44.499,158.150
C00581=1027.250,-115.175,414.368,166.743,44.502,158.151
C00582=1027.244,-115.425,414.377,166.740,44.504,158.151
C00583=1027.238,-115.675,414.386,166.738,44.507,158.151
C00584=1027.233,-115.925,414.394,166.734,44.509,158.151
C00585=1027.227,-116.174,414.403,166.732,44.511,158.151
C00586=1027.221,-116.424,414.412,166.728,44.514,158.151
C00587=1027.215,-116.710,414.422,166.725,44.516,158.151
C00588=1027.208,-116.996,414.431,166.722,44.519,158.151
C00589=1027.202,-117.282,414.442,166.718,44.522,158.152
C00590=1027.194,-117.568,414.452,166.715,44.525,158.152
C00591=1027.189,-117.818,414.461,166.712,44.528,158.152
C00592=1027.184,-118.068,414.469,166.709,44.530,158.152
C00593=1027.177,-118.318,414.477,166.706,44.533,158.152
C00594=1027.172,-118.567,414.486,166.703,44.535,158.152
C00595=1027.166,-118.817,414.495,166.700,44.537,158.153
C00596=1027.161,-119.067,414.504,166.697,44.540,158.153
C00597=1027.155,-119.317,414.512,166.694,44.542,158.153
C00598=1027.148,-119.566,414.521,166.692,44.545,158.153
C00599=1027.143,-119.816,414.530,166.688,44.548,158.153
C00600=1027.138,-120.066,414.538,166.686,44.550,158.153
C00601=1027.132,-120.316,414.547,166.682,44.553,158.153
C00602=1027.126,-120.565,414.555,166.680,44.555,158.154
C00603=1027.121,-120.815,414.563,166.676,44.557,158.154
C00604=1027.115,-121.066,414.572,166.674,44.559,158.154
C00605=1027.109,-121.315,414.582,166.670,44.562,158.154
C00606=1027.103,-121.564,414.589,166.668,44.565,158.154
C00607=1027.097,-121.814,414.598,166.664,44.567,158.154
C00608=1027.092,-122.064,414.607,166.662,44.570,158.154
C00609=1027.086,-122.314,414.615,166.659,44.573,158.155
C00610=1027.080,-122.564,414.623,166.656,44.575,158.155
C00611=1027.075,-122.814,414.632,166.653,44.577,158.155
C00612=1027.070,-123.063,414.640,166.650,44.579,158.155
C00613=1027.064,-123.313,414.648,166.646,44.582,158.155
C00614=1027.058,-123.563,414.657,166.644,44.585,158.155
C00615=1027.053,-123.813,414.666,166.640,44.587,158.155
C00616=1027.047,-124.062,414.674,166.638,44.590,158.156
C00617=1027.041,-124.313,414.682,166.635,44.592,158.156
C00618=1027.036,-124.563,414.691,166.632,44.595,158.156
C00619=1027.030,-124.812,414.699,166.630,44.597,158.156
C00620=1027.024,-125.062,414.707,166.626,44.600,158.156
C00621=1027.018,-125.312,414.716,166.624,44.602,158.156
C00622=1027.012,-125.561,414.724,166.620,44.605,158.156
C00623=1027.007,-125.811,414.733,166.618,44.608,158.157
C00624=1027.001,-126.061,414.740,166.614,44.610,158.157
C00625=1026.995,-126.311,414.749,166.612,44.613,158.157
C00626=1026.989,-126.560,414.757,166.608,44.615,158.157
C00627=1026.984,-126.810,414.766,166.606,44.617,158.157
C00628=1026.979,-127.060,414.774,166.602,44.620,158.157
C00629=1026.973,-127.310,414.781,166.600,44.623,158.158
C00630=1026.967,-127.560,414.790,166.597,44.626,158.158
C00631=1026.961,-127.810,414.798,166.594,44.628,158.158
C00632=1026.956,-128.058,414.807,166.591,44.631,158.158
C00633=1026.951,-128.308,414.815,166.588,44.633,158.158
C00634=1026.947,-128.558,414.825,166.585,44.634,158.158
C00635=1026.943,-128.808,414.835,166.582,44.634,158.158
C00636=1026.940,-129.057,414.846,166.580,44.635,158.158
C00637=1026.938,-129.307,414.858,166.577,44.635,158.157
C00638=1026.935,-129.557,414.870,166.575,44.635,158.157
C00639=1026.934,-129.806,414.881,166.573,44.634,158.157
C00640=1026.933,-130.057,414.895,166.570,44.632,158.156
C00641=1026.933,-130.306,414.908,166.569,44.630,158.156
C00642=1026.933,-130.556,414.923,166.566,44.628,158.155
C00643=1026.934,-130.806,414.938,166.564,44.625,158.154
C00644=1026.935,-131.056,414.953,166.563,44.622,158.154
C00645=1026.938,-131.306,414.969,166.560,44.618,158.153
C00646=1026.940,-131.555,414.985,166.559,44.614,158.152
C00647=1026.943,-131.805,415.003,166.557,44.609,158.151
C00648=1026.947,-132.056,415.020,166.556,44.604,158.150
C00649=1026.951,-132.305,415.038,166.555,44.598,158.149
C00650=1026.956,-132.555,415.058,166.553,44.592,158.148
C00651=1026.648,-132.580,414.738,166.504,44.850,158.186
C00652=1026.643,-132.331,414.718,166.507,44.857,158.188
C00653=1026.639,-132.081,414.700,166.507,44.863,158.189
C00654=1026.635,-131.831,414.682,166.509,44.867,158.190
C00655=1026.632,-131.581,414.666,166.511,44.872,158.191
C00656=1026.630,-131.331,414.649,166.512,44.877,158.192
C00657=1026.628,-131.082,414.632,166.515,44.881,158.193
C00658=1026.626,-130.831,414.617,166.516,44.884,158.193
C00659=1026.626,-130.581,414.602,166.518,44.887,158.194
C00660=1026.625,-130.332,414.589,166.520,44.889,158.194
C00661=1026.625,-130.082,414.575,166.522,44.891,158.195
C00662=1026.626,-129.832,414.561,166.524,44.892,158.195
C00663=1026.628,-129.582,414.549,166.527,44.893,158.196
C00664=1026.630,-129.333,414.538,166.529,44.894,158.196
C00665=1026.632,-129.082,414.526,166.532,44.894,158.196
C00666=1026.635,-128.833,414.515,166.534,44.893,158.197
C00667=1026.639,-128.583,414.505,166.537,44.892,158.197
C00668=1026.643,-128.334,414.495,166.540,44.891,158.197
C00669=1026.648,-128.085,414.486,166.542,44.889,158.197
C00670=1026.653,-127.835,414.478,166.545,44.887,158.197
C00671=1026.659,-127.585,414.470,166.548,44.884,158.196
C00672=1026.665,-127.336,414.462,166.551,44.881,158.196
C00673=1026.670,-127.085,414.453,166.554,44.878,158.196
C00674=1026.676,-126.836,414.445,166.558,44.876,158.196
C00675=1026.682,-126.586,414.436,166.560,44.873,158.196
C00676=1026.688,-126.337,414.429,166.564,44.870,158.196
C00677=1026.693,-126.086,414.421,166.566,44.868,158.195
C00678=1026.699,-125.836,414.412,166.570,44.866,158.195
C00679=1026.705,-125.587,414.404,166.572,44.863,158.195
C00680=1026.710,-125.337,414.396,166.575,44.860,158.195
C00681=1026.716,-125.088,414.388,166.578,44.857,158.195
C00682=1026.721,-124.838,414.379,166.581,44.855,158.195
C00683=1026.728,-124.588,414.371,166.584,44.852,158.195
C00684=1026.733,-124.338,414.362,166.587,44.849,158.194
C00685=1026.738,-124.088,414.354,166.590,44.847,158.194
C00686=1026.744,-123.838,414.345,166.593,44.845,158.194
C00687=1026.750,-123.588,414.337,166.596,44.842,158.194
C00688=1026.755,-123.339,414.329,166.599,44.839,158.194
C00689=1026.761,-123.089,414.320,166.602,44.837,158.194
C00690=1026.767,-122.839,414.312,166.605,44.834,158.193
C00691=1026.772,-122.589,414.303,166.607,44.831,158.193
C00692=1026.778,-122.339,414.295,166.611,44.829,158.193
C00693=1026.783,-122.090,414.286,166.613,44.827,158.193
C00694=1026.790,-121.840,414.278,166.617,44.824,158.193
C00695=1026.795,-121.590,414.270,166.619,44.822,158.193
C00696=1026.800,-121.340,414.261,166.623,44.819,158.193
C00697=1026.807,-121.091,414.252,166.625,44.816,158.192
C00698=1026.812,-120.841,414.244,166.629,44.814,158.192
C00699=1026.818,-120.591,414.235,166.631,44.811,158.192
C00700=1026.823,-120.341,414.226,166.635,44.809,158.192
C00701=1026.829,-120.091,414.219,166.637,44.806,158.192
C00702=1026.835,-119.842,414.210,166.640,44.803,158.192
C00703=1026.841,-119.591,414.201,166.643,44.801,158.192
C00704=1026.846,-119.342,414.192,166.646,44.799,158.192
C00705=1026.852,-119.093,414.184,166.649,44.796,158.191
C00706=1026.858,-118.842,414.175,166.652,44.794,158.191
C00707=1026.863,-118.593,414.167,166.655,44.791,158.191
C00708=1026.869,-118.343,414.158,166.658,44.788,158.191
C00709=1026.874,-118.093,414.149,166.661,44.786,158.191
C00710=1026.881,-117.844,414.141,166.664,44.783,158.191
C00711=1026.887,-117.593,414.132,166.667,44.781,158.190
C00712=1026.893,-117.308,414.122,166.670,44.778,158.190
C00713=1026.899,-117.021,414.112,166.673,44.775,158.190
C00714=1026.906,-116.736,414.102,166.677,44.772,158.190
C00715=1026.912,-116.450,414.092,166.680,44.769,158.190
C00716=1026.918,-116.200,414.084,166.684,44.767,158.190
C00717=1026.924,-115.950,414.075,166.686,44.764,158.190
C00718=1026.930,-115.701,414.066,166.690,44.762,158.190
C00719=1026.935,-115.450,414.057,166.692,44.759,158.189
C00720=1026.941,-115.201,414.049,166.696,44.756,158.189
C00721=1026.947,-114.951,414.039,166.698,44.754,158.189
C00722=1026.953,-114.702,414.031,166.702,44.752,158.189
C00723=1026.959,-114.451,414.022,166.704,44.750,158.189
C00724=1026.964,-114.202,414.013,166.708,44.747,158.189
C00725=1026.970,-113.952,414.004,166.710,44.744,158.188
C00726=1026.976,-113.703,413.995,166.714,44.742,158.188
C00727=1026.981,-113.453,413.987,166.716,44.739,158.188
C00728=1026.987,-113.202,413.978,166.720,44.737,158.188
C00729=1026.993,-112.953,413.969,166.722,44.734,158.188
C00730=1026.998,-112.703,413.960,166.726,44.732,158.188
C00731=1027.004,-112.454,413.950,166.728,44.729,158.188
C00732=1027.010,-112.203,413.942,166.732,44.727,158.188
C00733=1027.015,-111.954,413.932,166.734,44.725,158.187
C00734=1027.021,-111.704,413.924,166.738,44.722,158.187
C00735=1027.027,-111.455,413.914,166.740,44.720,158.187
C00736=1027.033,-111.204,413.906,166.743,44.717,158.187
C00737=1027.039,-110.955,413.896,166.746,44.715,158.187
C00738=1027.044,-110.705,413.887,166.749,44.712,158.187
C00739=1027.050,-110.455,413.878,166.752,44.710,158.187
C00740=1027.056,-110.205,413.869,166.754,44.707,158.186
C00741=1027.062,-109.955,413.860,166.758,44.705,158.186
C00742=1027.067,-109.706,413.851,166.760,44.702,158.186
C00743=1027.074,-109.456,413.842,166.764,44.700,158.186
C00744=1027.079,-109.207,413.834,166.766,44.698,158.186
C00745=1027.085,-108.957,413.824,166.770,44.695,158.186
C00746=1027.091,-108.706,413.815,166.772,44.693,158.186
C00747=1027.097,-108.457,413.806,166.776,44.690,158.186
C00748=1027.103,-108.207,413.797,166.778,44.688,158.185
C00749=1027.108,-107.958,413.788,166.782,44.685,158.185
C00750=1027.114,-107.708,413.779,166.785,44.683,158.185
C00751=1027.121,-107.458,413.769,166.788,44.680,158.185
C00752=1027.125,-107.208,413.760,166.791,44.678,158.185
C00753=1027.131,-106.958,413.750,166.794,44.675,158.185
C00754=1027.137,-106.709,413.741,166.797,44.673,158.185
C00755=1027.143,-106.459,413.732,166.799,44.671,158.184
C00756=1027.149,-106.209,413.723,166.803,44.668,158.184
C00757=1027.154,-105.960,413.714,166.805,44.666,158.184
C00758=1027.160,-105.709,413.705,166.809,44.664,158.184
C00759=1027.166,-105.460,413.695,166.811,44.662,158.184
C00760=1027.171,-105.210,413.685,166.815,44.659,158.184
C00761=1027.177,-104.960,413.676,166.817,44.657,158.184
C00762=1027.183,-104.711,413.667,166.821,44.654,158.184
C00763=1027.189,-104.461,413.658,166.823,44.652,158.184
C00764=1027.195,-104.211,413.648,166.826,44.649,158.183
C00765=1027.201,-103.962,413.639,166.829,44.647,158.183
C00766=1027.207,-103.712,413.630,166.832,44.644,158.183
C00767=1027.212,-103.462,413.620,166.835,44.642,158.183
C00768=1027.218,-103.212,413.611,166.838,44.640,158.183
C00769=1027.224,-102.963,413.601,166.841,44.637,158.183
C00770=1027.230,-102.713,413.592,166.844,44.635,158.183
C00771=1027.236,-102.463,413.582,166.847,44.633,158.183
C00772=1027.241,-102.213,413.573,166.850,44.631,158.182
C00773=1027.247,-101.963,413.563,166.852,44.628,158.182
C00774=1027.253,-101.713,413.554,166.856,44.626,158.182
C00775=1027.258,-101.464,413.545,166.858,44.624,158.182
C00776=1027.265,-101.178,413.534,166.862,44.621,158.182
C00777=1027.272,-100.891,413.523,166.865,44.618,158.182
C00778=1027.279,-100.605,413.511,166.869,44.615,158.182
C00779=1027.286,-100.319,413.501,166.872,44.612,158.181
C00780=1027.292,-100.069,413.491,166.875,44.610,158.181
C00781=1027.297,-99.820,413.482,166.878,44.608,158.181
C00782=1027.303,-99.570,413.472,166.881,44.606,158.181
C00783=1027.309,-99.320,413.462,166.884,44.603,158.181
C00784=1027.315,-99.070,413.452,166.887,44.601,158.181
C00785=1027.321,-98.820,413.444,166.890,44.599,158.181
C00786=1027.326,-98.570,413.434,166.893,44.596,158.181
C00787=1027.332,-98.320,413.424,166.896,44.594,158.181
C00788=1027.338,-98.071,413.415,166.899,44.591,158.180
C00789=1027.344,-97.821,413.405,166.901,44.589,158.180
C00790=1027.350,-97.571,413.395,166.905,44.587,158.180
C00791=1027.356,-97.322,413.385,166.907,44.584,158.180
C00792=1027.361,-97.072,413.375,166.911,44.582,158.180
C00793=1027.367,-96.822,413.365,166.914,44.580,158.180
C00794=1027.373,-96.572,413.356,166.916,44.578,158.180
C00795=1027.379,-96.322,413.346,166.920,44.575,158.180
C00796=1027.384,-96.073,413.336,166.922,44.573,158.179
C00797=1027.390,-95.823,413.326,166.925,44.571,158.179
C00798=1027.396,-95.573,413.317,166.928,44.568,158.179
C00799=1027.402,-95.324,413.306,166.931,44.567,158.179
C00800=1027.408,-95.074,413.296,166.934,44.564,158.179
C00801=1027.413,-94.824,413.286,166.937,44.562,158.179
C00802=1027.419,-94.575,413.277,166.939,44.560,158.179
C00803=1027.424,-94.325,413.267,166.943,44.558,158.179
C00804=1027.431,-94.076,413.256,166.946,44.556,158.179
C00805=1027.436,-93.825,413.246,166.948,44.554,158.179
C00806=1027.442,-93.576,413.237,166.952,44.551,158.178
C00807=1027.448,-93.326,413.226,166.954,44.549,158.178
C00808=1027.454,-93.076,413.217,166.957,44.547,158.178
C00809=1027.460,-92.826,413.206,166.961,44.545,158.178
C00810=1027.465,-92.577,413.197,166.963,44.542,158.178
C00811=1027.471,-92.327,413.187,166.967,44.540,158.178
C00812=1027.477,-92.078,413.176,166.969,44.538,158.178
C00813=1027.483,-91.828,413.166,166.972,44.535,158.178
C00814=1027.489,-91.578,413.157,166.975,44.533,158.178
C00815=1027.494,-91.328,413.147,166.978,44.531,158.177
C00816=1027.501,-91.079,413.136,166.980,44.529,158.177
C00817=1027.506,-90.829,413.126,166.984,44.526,158.177
C00818=1027.512,-90.579,413.116,166.986,44.524,158.177
C00819=1027.518,-90.329,413.106,166.990,44.522,158.177
C00820=1027.524,-90.079,413.096,166.992,44.520,158.177
C00821=1027.530,-89.829,413.086,166.995,44.518,158.177
C00822=1027.536,-89.580,413.076,166.999,44.515,158.177
C00823=1027.542,-89.330,413.065,167.001,44.513,158.177
C00824=1027.548,-89.080,413.056,167.004,44.511,158.176
C00825=1027.554,-88.831,413.045,167.007,44.509,158.176
C00826=1027.559,-88.581,413.035,167.010,44.507,158.176
C00827=1027.565,-88.331,413.025,167.013,44.504,158.176
C00828=1027.571,-88.081,413.014,167.016,44.502,158.176
C00829=1027.577,-87.832,413.005,167.019,44.500,158.176
C00830=1027.583,-87.582,412.994,167.022,44.498,158.176
C00831=1027.589,-87.332,412.984,167.025,44.495,158.176
C00832=1027.595,-87.083,412.974,167.027,44.493,158.175
C00833=1027.601,-86.833,412.964,167.031,44.491,158.175
C00834=1027.607,-86.584,412.953,167.033,44.488,158.175
C00835=1027.613,-86.334,412.943,167.037,44.486,158.175
C00836=1027.619,-86.084,412.933,167.039,44.484,158.175
C00837=1027.625,-85.834,412.923,167.042,44.482,158.175
C00838=1027.630,-85.585,412.912,167.045,44.479,158.175
C00839=1027.636,-85.335,412.902,167.048,44.477,158.175
C00840=1027.643,-85.051,412.891,167.052,44.475,158.175
C00841=1027.650,-84.766,412.879,167.055,44.472,158.174
C00842=1027.657,-84.483,412.866,167.059,44.470,158.174
C00843=1027.664,-84.198,412.855,167.061,44.467,158.174
C00844=1027.669,-83.948,412.845,167.065,44.465,158.174
C00845=1027.676,-83.699,412.835,167.067,44.463,158.174
C00846=1027.681,-83.449,412.825,167.071,44.460,158.174
C00847=1027.688,-83.200,412.814,167.073,44.458,158.174
C00848=1027.694,-82.950,412.803,167.076,44.456,158.174
C00849=1027.700,-82.699,412.793,167.079,44.453,158.173
C00850=1027.706,-82.450,412.783,167.082,44.451,158.173
C00851=1027.712,-82.200,412.772,167.084,44.449,158.173
C00852=1027.718,-81.951,412.762,167.088,44.446,158.173
C00853=1027.724,-81.701,412.751,167.090,44.445,158.173
C00854=1027.730,-81.452,412.742,167.094,44.442,158.173
C00855=1027.736,-81.201,412.730,167.096,44.440,158.173
C00856=1027.742,-80.952,412.720,167.099,44.438,158.173
C00857=1027.748,-80.702,412.710,167.103,44.436,158.173
C00858=1027.754,-80.453,412.699,167.105,44.434,158.172
C00859=1027.760,-80.203,412.689,167.108,44.431,158.172
C00860=1027.766,-79.953,412.678,167.111,44.429,158.172
C00861=1027.772,-79.703,412.667,167.114,44.427,158.172
C00862=1027.778,-79.454,412.657,167.117,44.425,158.172
C00863=1027.783,-79.204,412.646,167.120,44.422,158.172
C00864=1027.790,-78.954,412.636,167.123,44.420,158.172
C00865=1027.796,-78.704,412.625,167.125,44.418,158.172
C00866=1027.802,-78.455,412.614,167.129,44.416,158.172
C00867=1027.808,-78.205,412.603,167.131,44.414,158.171
C00868=1027.813,-77.956,412.592,167.134,44.412,158.171
C00869=1027.819,-77.706,412.582,167.138,44.410,158.171
C00870=1027.826,-77.456,412.571,167.140,44.407,158.171
C00871=1027.832,-77.206,412.561,167.143,44.405,158.171
C00872=1027.837,-76.957,412.550,167.145,44.403,158.171
C00873=1027.843,-76.707,412.539,167.149,44.401,158.171
C00874=1027.849,-76.457,412.528,167.152,44.399,158.171
C00875=1027.855,-76.208,412.517,167.154,44.397,158.171
C00876=1027.861,-75.958,412.507,167.158,44.395,158.170
C00877=1027.867,-75.708,412.496,167.160,44.393,158.170
C00878=1027.873,-75.458,412.485,167.163,44.391,158.170
C00879=1027.879,-75.209,412.474,167.166,44.389,158.170
C00880=1027.885,-74.959,412.463,167.169,44.387,158.170
C00881=1027.891,-74.709,412.452,167.172,44.385,158.170
C00882=1027.897,-74.459,412.441,167.175,44.382,158.170
C00883=1027.903,-74.210,412.431,167.178,44.380,158.170
C00884=1027.908,-73.960,412.419,167.180,44.378,158.170
C00885=1027.915,-73.710,412.408,167.183,44.376,158.170
C00886=1027.921,-73.461,412.397,167.187,44.374,158.169
C00887=1027.926,-73.211,412.386,167.189,44.372,158.169
C00888=1027.933,-72.961,412.375,167.192,44.370,158.169
C00889=1027.938,-72.712,412.364,167.194,44.368,158.169
C00890=1027.944,-72.462,412.353,167.197,44.366,158.169
C00891=1027.950,-72.212,412.341,167.201,44.364,158.169
C00892=1027.956,-71.963,412.330,167.203,44.362,158.169
C00893=1027.961,-71.713,412.319,167.206,44.360,158.169
C00894=1027.967,-71.464,412.308,167.208,44.358,158.169
C00895=1027.974,-71.214,412.297,167.212,44.356,158.169
C00896=1027.979,-70.964,412.286,167.215,44.354,158.169
C00897=1027.985,-70.715,412.275,167.217,44.352,158.168
C00898=1027.991,-70.464,412.263,167.220,44.350,158.168
C00899=1027.997,-70.215,412.252,167.224,44.348,158.168
C00900=1028.003,-69.965,412.240,167.226,44.346,158.168
C00901=1028.009,-69.716,412.230,167.229,44.344,158.168
C00902=1028.015,-69.466,412.219,167.231,44.342,158.168
C00903=1028.021,-69.216,412.207,167.234,44.340,158.168
C00904=1028.027,-68.935,412.194,167.238,44.338,158.168
C00905=1028.033,-68.653,412.181,167.241,44.336,158.168
C00906=1028.041,-68.370,412.169,167.244,44.334,158.168
C00907=1028.047,-68.088,412.156,167.247,44.331,158.168
C00908=1028.053,-67.838,412.145,167.250,44.329,158.167
C00909=1028.059,-67.589,412.134,167.254,44.327,158.167
C00910=1028.065,-67.340,412.123,167.256,44.325,158.167
C00911=1028.071,-67.089,412.111,167.259,44.323,158.167
C00912=1028.077,-66.840,412.099,167.261,44.321,158.167
C00913=1028.083,-66.590,412.088,167.264,44.319,158.167
C00914=1028.089,-66.341,412.077,167.268,44.317,158.167
C00915=1028.095,-66.090,412.066,167.270,44.315,158.167
C00916=1028.101,-65.842,412.054,167.273,44.313,158.167
C00917=1028.107,-65.591,412.043,167.276,44.311,158.167
C00918=1028.113,-65.342,412.032,167.279,44.309,158.167
C00919=1028.119,-65.093,412.020,167.282,44.307,158.167
C00920=1028.125,-64.843,412.009,167.284,44.305,158.166
C00921=1028.131,-64.593,411.998,167.287,44.303,158.166
C00922=1028.137,-64.343,411.985,167.290,44.301,158.166
C00923=1028.142,-64.094,411.974,167.293,44.299,158.166
C00924=1028.149,-63.844,411.963,167.296,44.297,158.166
C00925=1028.155,-63.595,411.952,167.299,44.295,158.166
C00926=1028.161,-63.344,411.940,167.301,44.293,158.166
C00927=1028.166,-63.095,411.928,167.305,44.291,158.166
C00928=1028.173,-62.845,411.917,167.307,44.289,158.166
C00929=1028.179,-62.596,411.905,167.310,44.287,158.166
C00930=1028.185,-62.346,411.894,167.313,44.285,158.165
C00931=1028.192,-62.096,411.883,167.316,44.283,158.165
C00932=1028.197,-61.847,411.871,167.319,44.281,158.165
C00933=1028.203,-61.596,411.859,167.321,44.279,158.165
C00934=1028.209,-61.348,411.848,167.324,44.277,158.165
C00935=1028.216,-61.097,411.837,167.326,44.275,158.165
C00936=1028.222,-60.848,411.825,167.330,44.273,158.165
C00937=1028.227,-60.598,411.813,167.333,44.271,158.165
C00938=1028.233,-60.349,411.802,167.335,44.269,158.165
C00939=1028.240,-60.099,411.790,167.338,44.267,158.165
C00940=1028.246,-59.849,411.778,167.342,44.265,158.164
C00941=1028.252,-59.600,411.768,167.344,44.263,158.164
C00942=1028.258,-59.350,411.755,167.347,44.261,158.164
C00943=1028.264,-59.100,411.744,167.349,44.259,158.164
C00944=1028.270,-58.851,411.732,167.352,44.257,158.164
C00945=1028.277,-58.601,411.721,167.356,44.255,158.164
C00946=1028.283,-58.352,411.709,167.358,44.253,158.164
C00947=1028.289,-58.102,411.697,167.361,44.251,158.164
C00948=1028.295,-57.852,411.686,167.364,44.249,158.164
C00949=1028.301,-57.603,411.674,167.367,44.247,158.164
C00950=1028.307,-57.353,411.663,167.370,44.244,158.163
C00951=1028.313,-57.103,411.650,167.372,44.242,158.163
C00952=1028.319,-56.854,411.639,167.375,44.240,158.163
C00953=1028.326,-56.604,411.627,167.377,44.238,158.163
C00954=1028.332,-56.354,411.615,167.381,44.236,158.163
C00955=1028.337,-56.104,411.604,167.384,44.234,158.163
C00956=1028.344,-55.855,411.592,167.386,44.232,158.163
C00957=1028.351,-55.605,411.580,167.389,44.231,158.163
C00958=1028.356,-55.356,411.569,167.393,44.228,158.163
C00959=1028.362,-55.106,411.556,167.395,44.227,158.163
C00960=1028.369,-54.856,411.545,167.398,44.225,158.162
C00961=1028.375,-54.607,411.534,167.400,44.222,158.162
C00962=1028.381,-54.357,411.522,167.403,44.220,158.162
C00963=1028.387,-54.107,411.509,167.406,44.218,158.162
C00964=1028.394,-53.858,411.497,167.409,44.216,158.162
C00965=1028.399,-53.608,411.486,167.412,44.214,158.162
C00966=1028.406,-53.359,411.474,167.414,44.212,158.162
C00967=1028.412,-53.109,411.462,167.418,44.210,158.162
C00968=1028.419,-52.828,411.449,167.420,44.207,158.161
C00969=1028.427,-52.547,411.436,167.424,44.205,158.161
C00970=1028.433,-52.266,411.422,167.427,44.203,158.161
C00971=1028.441,-51.986,411.409,167.430,44.200,158.161
C00972=1028.449,-51.634,411.392,167.434,44.197,158.161
C00973=1028.458,-51.282,411.376,167.438,44.195,158.161
C00974=1028.464,-51.032,411.364,167.440,44.193,158.161
C00975=1028.470,-50.783,411.352,167.443,44.191,158.161
C00976=1028.477,-50.533,411.340,167.447,44.189,158.160
C00977=1028.483,-50.283,411.327,167.449,44.187,158.160
C00978=1028.488,-50.034,411.315,167.452,44.185,158.160
C00979=1028.495,-49.784,411.303,167.454,44.183,158.160
C00980=1028.501,-49.534,411.290,167.457,44.182,158.160
C00981=1028.507,-49.285,411.278,167.460,44.180,158.160
C00982=1028.513,-49.035,411.266,167.463,44.178,158.160
C00983=1028.519,-48.786,411.254,167.465,44.176,158.160
C00984=1028.525,-48.536,411.242,167.469,44.174,158.160
C00985=1028.531,-48.286,411.229,167.471,44.172,158.160
C00986=1028.537,-48.036,411.217,167.474,44.170,158.160
C00987=1028.544,-47.787,411.205,167.477,44.168,158.159
C00988=1028.549,-47.538,411.193,167.480,44.167,158.159
C00989=1028.555,-47.288,411.180,167.482,44.165,158.159
C00990=1028.561,-47.038,411.168,167.485,44.163,158.159
C00991=1028.567,-46.788,411.155,167.487,44.161,158.159
C00992=1028.573,-46.538,411.143,167.491,44.159,158.159
C00993=1028.579,-46.290,411.131,167.494,44.157,158.159
C00994=1028.585,-46.040,411.119,167.496,44.155,158.159
C00995=1028.591,-45.790,411.106,167.499,44.153,158.159
C00996=1028.598,-45.540,411.094,167.501,44.151,158.159
C00997=1028.604,-45.290,411.082,167.504,44.149,158.159
C00998=1028.610,-45.040,411.069,167.507,44.147,158.158
C00999=1028.617,-44.792,411.056,167.510,44.146,158.158
C01000=1028.622,-44.542,411.044,167.512,44.144,158.158
C01001=1028.628,-44.292,411.032,167.516,44.142,158.158
C01002=1028.634,-44.043,411.020,167.518,44.140,158.158
C01003=1028.640,-43.793,411.007,167.521,44.138,158.158
C01004=1028.646,-43.543,410.995,167.524,44.136,158.158
C01005=1028.653,-43.294,410.983,167.526,44.134,158.158
C01006=1028.659,-43.044,410.969,167.529,44.132,158.158
C01007=1028.665,-42.794,410.957,167.531,44.130,158.158
C01008=1028.672,-42.545,410.945,167.534,44.128,158.158
C01009=1028.678,-42.295,410.932,167.537,44.127,158.157
C01010=1028.683,-42.045,410.920,167.540,44.124,158.157
C01011=1028.690,-41.796,410.907,167.543,44.122,158.157
C01012=1028.696,-41.546,410.895,167.546,44.121,158.157
C01013=1028.702,-41.297,410.882,167.548,44.119,158.157
C01014=1028.708,-41.048,410.870,167.551,44.117,158.157
C01015=1028.715,-40.798,410.857,167.554,44.115,158.157
C01016=1028.720,-40.548,410.845,167.556,44.114,158.157
C01017=1028.727,-40.299,410.833,167.559,44.112,158.157
C01018=1028.733,-40.049,410.820,167.562,44.110,158.157
C01019=1028.739,-39.800,410.807,167.565,44.108,158.157
C01020=1028.746,-39.550,410.795,167.568,44.106,158.156
C01021=1028.752,-39.300,410.782,167.570,44.104,158.156
C01022=1028.758,-39.051,410.769,167.573,44.102,158.156
C01023=1028.764,-38.801,410.756,167.576,44.100,158.156
C01024=1028.770,-38.551,410.744,167.578,44.098,158.156
C01025=1028.776,-38.302,410.731,167.581,44.097,158.156
C01026=1028.782,-38.052,410.718,167.584,44.095,158.156
C01027=1028.788,-37.802,410.706,167.586,44.093,158.156
C01028=1028.795,-37.553,410.693,167.589,44.091,158.156
C01029=1028.801,-37.303,410.680,167.592,44.089,158.156
C01030=1028.809,-36.949,410.661,167.595,44.087,158.156
C01031=1028.818,-36.595,410.644,167.600,44.084,158.155
C01032=1028.827,-36.241,410.625,167.603,44.082,158.155
C01033=1028.836,-35.887,410.607,167.607,44.079,158.155
C01034=1028.842,-35.637,410.594,167.609,44.077,158.155
C01035=1028.848,-35.387,410.581,167.613,44.075,158.155
C01036=1028.854,-35.138,410.568,167.616,44.074,158.155
C01037=1028.860,-34.888,410.556,167.618,44.072,158.155
C01038=1028.866,-34.639,410.542,167.621,44.070,158.155
C01039=1028.872,-34.389,410.530,167.624,44.068,158.155
C01040=1028.878,-34.140,410.517,167.626,44.066,158.155
C01041=1028.884,-33.890,410.504,167.629,44.064,158.154
C01042=1028.890,-33.641,410.491,167.632,44.063,158.154
C01043=1028.897,-33.391,410.477,167.634,44.061,158.154
C01044=1028.903,-33.141,410.465,167.637,44.059,158.154
C01045=1028.909,-32.892,410.451,167.640,44.057,158.154
C01046=1028.915,-32.642,410.439,167.642,44.055,158.154
C01047=1028.921,-32.392,410.425,167.645,44.053,158.154
C01048=1028.927,-32.143,410.413,167.647,44.051,158.154
C01049=1028.933,-31.893,410.400,167.650,44.050,158.154
C01050=1028.940,-31.644,410.386,167.653,44.048,158.154
C01051=1028.946,-31.394,410.374,167.655,44.046,158.154
C01052=1028.952,-31.144,410.360,167.658,44.044,158.153
C01053=1028.959,-30.895,410.347,167.661,44.043,158.153
C01054=1028.964,-30.645,410.334,167.663,44.041,158.153
C01055=1028.971,-30.396,410.321,167.666,44.039,158.153
C01056=1028.977,-30.147,410.308,167.669,44.037,158.153
C01057=1028.983,-29.897,410.295,167.671,44.036,158.153
C01058=1028.989,-29.647,410.282,167.674,44.034,158.153
C01059=1028.996,-29.397,410.268,167.677,44.032,158.153
C01060=1029.002,-29.148,410.256,167.679,44.030,158.153
C01061=1029.008,-28.898,410.243,167.683,44.028,158.153
C01062=1029.014,-28.649,410.229,167.686,44.026,158.153
C01063=1029.020,-28.399,410.217,167.688,44.024,158.152
C01064=1029.027,-28.149,410.203,167.691,44.022,158.152
C01065=1029.033,-27.900,410.190,167.693,44.020,158.152
C01066=1029.039,-27.651,410.177,167.696,44.019,158.152
C01067=1029.045,-27.401,410.164,167.699,44.017,158.152
C01068=1029.051,-27.151,410.151,167.701,44.015,158.152
C01069=1029.058,-26.902,410.137,167.704,44.013,158.152
C01070=1029.064,-26.652,410.124,167.707,44.011,158.152
C01071=1029.071,-26.403,410.111,167.710,44.010,158.152
C01072=1029.076,-26.153,410.097,167.712,44.008,158.152
C01073=1029.082,-25.904,410.084,167.715,44.006,158.152
C01074=1029.089,-25.654,410.070,167.717,44.004,158.151
C01075=1029.095,-25.404,410.057,167.719,44.003,158.151
C01076=1029.101,-25.155,410.043,167.722,44.001,158.151
C01077=1029.107,-24.905,410.030,167.724,43.999,158.151
C01078=1029.114,-24.655,410.016,167.727,43.997,158.151
C01079=1029.120,-24.406,410.003,167.730,43.996,158.151
C01080=1029.125,-24.157,409.989,167.733,43.994,158.151
C01081=1029.132,-23.907,409.976,167.735,43.992,158.151
C01082=1029.138,-23.657,409.963,167.738,43.990,158.151
C01083=1029.143,-23.407,409.949,167.741,43.989,158.151
C01084=1029.150,-23.158,409.936,167.743,43.987,158.151
C01085=1029.156,-22.909,409.923,167.746,43.985,158.150
C01086=1029.163,-22.659,409.909,167.748,43.983,158.150
C01087=1029.168,-22.409,409.895,167.751,43.982,158.150
C01088=1029.174,-22.160,409.882,167.754,43.980,158.150
C01089=1029.181,-21.910,409.868,167.757,43.978,158.150
C01090=1029.187,-21.661,409.855,167.759,43.976,158.150
C01091=1029.193,-21.411,409.841,167.762,43.975,158.150
C01092=1029.199,-21.162,409.828,167.765,43.973,158.150
C01093=1029.206,-20.912,409.814,167.767,43.971,158.150
C01094=1029.213,-20.631,409.799,167.770,43.969,158.150
C01095=1029.220,-20.350,409.783,167.773,43.967,158.150
C01096=1029.227,-20.068,409.768,167.776,43.965,158.150
C01097=1029.234,-19.787,409.753,167.779,43.964,158.149
C01098=1029.240,-19.538,409.739,167.781,43.962,158.149
C01099=1029.246,-19.288,409.725,167.784,43.960,158.149
C01100=1029.253,-19.038,409.712,167.787,43.958,158.149
C01101=1029.259,-18.789,409.699,167.789,43.956,158.149
C01102=1029.264,-18.539,409.685,167.792,43.955,158.149
C01103=1029.271,-18.290,409.671,167.795,43.953,158.149
C01104=1029.277,-18.040,409.658,167.797,43.951,158.149
C01105=1029.284,-17.791,409.643,167.800,43.949,158.149
C01106=1029.290,-17.541,409.630,167.803,43.947,158.148
C01107=1029.296,-17.292,409.616,167.805,43.945,158.148
C01108=1029.303,-17.042,409.603,167.808,43.944,158.148
C01109=1029.308,-16.793,409.589,167.811,43.942,158.148
C01110=1029.315,-16.543,409.575,167.813,43.940,158.148
C01111=1029.321,-16.293,409.562,167.816,43.938,158.148
C01112=1029.327,-16.044,409.547,167.818,43.936,158.148
C01113=1029.334,-15.794,409.534,167.821,43.934,158.148
C01114=1029.340,-15.545,409.520,167.824,43.933,158.148
C01115=1029.346,-15.295,409.506,167.825,43.931,158.148
C01116=1029.353,-15.046,409.493,167.828,43.930,158.148
C01117=1029.359,-14.796,409.478,167.831,43.928,158.148
C01118=1029.364,-14.546,409.464,167.834,43.926,158.147
C01119=1029.371,-14.297,409.451,167.836,43.924,158.147
C01120=1029.377,-14.047,409.436,167.839,43.923,158.147
C01121=1029.383,-13.798,409.423,167.842,43.921,158.147
C01122=1029.389,-13.548,409.408,167.844,43.919,158.147
C01123=1029.396,-13.299,409.394,167.847,43.918,158.147
C01124=1029.401,-13.050,409.381,167.850,43.916,158.147
C01125=1029.408,-12.800,409.367,167.851,43.915,158.147
C01126=1029.414,-12.551,409.352,167.854,43.913,158.147
C01127=1029.420,-12.300,409.338,167.857,43.911,158.147
C01128=1029.426,-12.051,409.325,167.859,43.910,158.147
C01129=1029.433,-11.802,409.310,167.862,43.908,158.146
C01130=1029.439,-11.552,409.297,167.865,43.906,158.146
C01131=1029.445,-11.303,409.282,167.867,43.904,158.146
C01132=1029.451,-11.053,409.268,167.870,43.903,158.146
C01133=1029.457,-10.803,409.254,167.873,43.901,158.146
C01134=1029.463,-10.554,409.240,167.874,43.899,158.146
C01135=1029.470,-10.304,409.226,167.877,43.898,158.146
C01136=1029.476,-10.055,409.211,167.880,43.896,158.146
C01137=1029.483,-9.805,409.198,167.882,43.894,158.146
C01138=1029.488,-9.556,409.183,167.885,43.892,158.146
C01139=1029.495,-9.306,409.170,167.888,43.891,158.146
C01140=1029.501,-9.057,409.156,167.890,43.889,158.146
C01141=1029.507,-8.807,409.141,167.893,43.887,158.145
C01142=1029.513,-8.558,409.127,167.896,43.885,158.145
C01143=1029.520,-8.308,409.113,167.898,43.884,158.145
C01144=1029.526,-8.059,409.099,167.900,43.882,158.145
C01145=1029.532,-7.809,409.084,167.903,43.880,158.145
C01146=1029.538,-7.560,409.070,167.905,43.878,158.145
C01147=1029.545,-7.310,409.056,167.908,43.877,158.145
C01148=1029.551,-7.060,409.042,167.911,43.875,158.145
C01149=1029.558,-6.811,409.028,167.913,43.873,158.145
C01150=1029.564,-6.561,409.014,167.916,43.871,158.145
C01151=1029.569,-6.312,408.999,167.919,43.870,158.145
C01152=1029.576,-6.063,408.985,167.921,43.868,158.144
C01153=1029.582,-5.813,408.971,167.923,43.867,158.144
C01154=1029.589,-5.564,408.956,167.926,43.865,158.144
C01155=1029.595,-5.314,408.942,167.928,43.863,158.144
C01156=1029.601,-5.065,408.928,167.931,43.862,158.144
C01157=1029.608,-4.815,408.914,167.934,43.860,158.144
C01158=1029.615,-4.533,408.897,167.936,43.858,158.144
C01159=1029.622,-4.249,408.882,167.939,43.856,158.144
C01160=1029.629,-3.967,408.866,167.943,43.854,158.144
C01161=1029.636,-3.684,408.849,167.945,43.852,158.143
C01162=1029.642,-3.433,408.834,167.948,43.850,158.143
C01163=1029.648,-3.185,408.820,167.951,43.849,158.143
C01164=1029.654,-2.935,408.805,167.952,43.847,158.143
C01165=1029.660,-2.686,408.790,167.955,43.845,158.143
C01166=1029.666,-2.436,408.776,167.958,43.844,158.143
C01167=1029.673,-2.186,408.761,167.961,43.842,158.143
C01168=1029.678,-1.937,408.746,167.963,43.841,158.143
C01169=1029.685,-1.687,408.731,167.965,43.839,158.143
C01170=1029.691,-1.439,408.718,167.968,43.837,158.143
C01171=1029.697,-1.188,408.703,167.970,43.836,158.143
C01172=1029.704,-0.939,408.688,167.973,43.834,158.143
C01173=1029.710,-0.690,408.674,167.976,43.833,158.143
C01174=1029.716,-0.440,408.659,167.977,43.831,158.142
C01175=1029.722,-0.191,408.644,167.980,43.829,158.142
C01176=1029.728,0.059,408.630,167.983,43.828,158.142
C01177=1029.734,0.309,408.615,167.986,43.826,158.142
C01178=1029.740,0.558,408.600,167.988,43.825,158.142
C01179=1029.746,0.807,408.586,167.990,43.823,158.142
C01180=1029.753,1.057,408.571,167.993,43.821,158.142
C01181=1029.759,1.306,408.556,167.995,43.820,158.142
C01182=1029.765,1.556,408.541,167.998,43.818,158.142
C01183=1029.771,1.805,408.526,168.001,43.816,158.142
C01184=1029.777,2.056,408.512,168.003,43.815,158.142
C01185=1029.783,2.304,408.497,168.005,43.813,158.142
C01186=1029.790,2.554,408.482,168.008,43.811,158.141
C01187=1029.796,2.804,408.467,168.011,43.810,158.141
C01188=1029.802,3.053,408.453,168.013,43.808,158.141
C01189=1029.808,3.302,408.438,168.015,43.807,158.141
C01190=1029.815,3.552,408.423,168.018,43.805,158.141
C01191=1029.820,3.801,408.408,168.020,43.804,158.141
C01192=1029.827,4.051,408.393,168.023,43.802,158.141
C01193=1029.833,4.300,408.378,168.026,43.800,158.141
C01194=1029.839,4.550,408.364,168.027,43.799,158.141
C01195=1029.846,4.799,408.350,168.030,43.797,158.141
C01196=1029.852,5.048,408.335,168.033,43.796,158.141
C01197=1029.859,5.298,408.320,168.035,43.794,158.140
C01198=1029.865,5.548,408.305,168.038,43.792,158.140
C01199=1029.871,5.797,408.290,168.040,43.791,158.140
C01200=1029.877,6.046,408.275,168.042,43.789,158.140
C01201=1029.884,6.296,408.260,168.045,43.787,158.140
C01202=1029.890,6.546,408.245,168.048,43.786,158.140
C01203=1029.896,6.795,408.230,168.051,43.784,158.140
C01204=1029.902,7.044,408.216,168.052,43.782,158.140
C01205=1029.909,7.294,408.201,168.055,43.780,158.140
C01206=1029.915,7.543,408.186,168.058,43.779,158.140
C01207=1029.921,7.793,408.171,168.060,43.777,158.140
C01208=1029.928,8.043,408.156,168.063,43.775,158.139
C01209=1029.934,8.292,408.141,168.065,43.774,158.139
C01210=1029.940,8.541,408.126,168.067,43.772,158.139
C01211=1029.946,8.791,408.111,168.070,43.770,158.139
C01212=1029.953,9.041,408.097,168.073,43.769,158.139
C01213=1029.959,9.290,408.081,168.075,43.767,158.139
C01214=1029.965,9.539,408.066,168.078,43.765,158.139
C01215=1029.972,9.788,408.051,168.080,43.764,158.139
C01216=1029.978,10.038,408.036,168.082,43.762,158.139
C01217=1029.984,10.288,408.021,168.085,43.761,158.139
C01218=1029.991,10.537,408.007,168.088,43.759,158.138
C01219=1029.997,10.787,407.992,168.090,43.757,158.138
C01220=1030.004,11.036,407.976,168.092,43.755,158.138
C01221=1030.010,11.285,407.961,168.095,43.754,158.138
C01222=1030.017,11.570,407.944,168.097,43.752,158.138
C01223=1030.024,11.855,407.927,168.101,43.750,158.138
C01224=1030.031,12.140,407.909,168.104,43.748,158.138
C01225=1030.039,12.425,407.893,168.106,43.746,158.138
C01226=1030.045,12.674,407.878,168.109,43.744,158.138
C01227=1030.052,12.924,407.863,168.112,43.742,158.137
C01228=1030.058,13.173,407.847,168.113,43.741,158.137
C01229=1030.063,13.422,407.832,168.116,43.739,158.137
C01230=1030.070,13.672,407.817,168.119,43.738,158.137
C01231=1030.076,13.922,407.802,168.121,43.736,158.137
C01232=1030.083,14.171,407.786,168.123,43.734,158.137
C01233=1030.089,14.420,407.771,168.126,43.733,158.137
C01234=1030.095,14.670,407.756,168.128,43.731,158.137
C01235=1030.102,14.919,407.740,168.131,43.730,158.137
C01236=1030.108,15.169,407.725,168.133,43.728,158.137
C01237=1030.114,15.419,407.710,168.135,43.726,158.136
C01238=1030.120,15.668,407.694,168.138,43.725,158.137
C01239=1030.127,15.918,407.679,168.141,43.723,158.136
C01240=1030.133,16.167,407.664,168.142,43.721,158.136
C01241=1030.138,16.416,407.648,168.145,43.720,158.136
C01242=1030.145,16.666,407.633,168.148,43.718,158.136
C01243=1030.152,16.915,407.618,168.150,43.716,158.136
C01244=1030.158,17.164,407.603,168.152,43.715,158.136
C01245=1030.164,17.414,407.586,168.155,43.713,158.136
C01246=1030.170,17.663,407.572,168.158,43.712,158.136
C01247=1030.177,17.913,407.557,168.160,43.710,158.136
C01248=1030.183,18.162,407.540,168.162,43.709,158.135
C01249=1030.189,18.412,407.525,168.165,43.707,158.135
C01250=1030.196,18.661,407.510,168.167,43.705,158.135
C01251=1030.201,18.911,407.494,168.170,43.704,158.135
C01252=1030.208,19.160,407.479,168.172,43.702,158.135
C01253=1030.214,19.410,407.464,168.175,43.701,158.135
C01254=1030.221,19.659,407.448,168.177,43.699,158.135
C01255=1030.227,19.909,407.432,168.179,43.698,158.135
C01256=1030.233,20.158,407.417,168.182,43.696,158.135
C01257=1030.239,20.408,407.401,168.184,43.694,158.135
C01258=1030.246,20.657,407.386,168.187,43.693,158.135
C01259=1030.251,20.907,407.370,168.189,43.691,158.134
C01260=1030.258,21.156,407.354,168.191,43.690,158.135
C01261=1030.264,21.405,407.338,168.194,43.688,158.134
C01262=1030.270,21.655,407.323,168.196,43.686,158.134
C01263=1030.277,21.904,407.307,168.199,43.685,158.134
C01264=1030.283,22.154,407.292,168.201,43.683,158.134
C01265=1030.289,22.403,407.276,168.204,43.681,158.134
C01266=1030.295,22.653,407.261,168.206,43.680,158.134
C01267=1030.302,22.902,407.245,168.208,43.678,158.134
C01268=1030.308,23.151,407.229,168.211,43.677,158.134
C01269=1030.314,23.401,407.214,168.213,43.676,158.134
C01270=1030.320,23.650,407.198,168.215,43.674,158.133
C01271=1030.327,23.899,407.182,168.218,43.672,158.133
C01272=1030.332,24.149,407.166,168.221,43.671,158.133
C01273=1030.339,24.398,407.151,168.222,43.669,158.133
C01274=1030.346,24.647,407.135,168.225,43.668,158.133
C01275=1030.351,24.897,407.120,168.228,43.666,158.133
C01276=1030.358,25.146,407.104,168.229,43.664,158.133
C01277=1030.364,25.396,407.088,168.232,43.663,158.133
C01278=1030.371,25.646,407.072,168.235,43.661,158.133
C01279=1030.377,25.895,407.056,168.238,43.659,158.133
C01280=1030.384,26.144,407.040,168.239,43.658,158.133
C01281=1030.390,26.394,407.024,168.242,43.656,158.132
C01282=1030.396,26.643,407.009,168.245,43.654,158.132
C01283=1030.402,26.893,406.993,168.246,43.653,158.132
C01284=1030.409,27.142,406.977,168.249,43.651,158.132
C01285=1030.415,27.391,406.961,168.252,43.650,158.132
C01286=1030.422,27.678,406.943,168.255,43.648,158.132
C01287=1030.429,27.963,406.925,168.257,43.646,158.132
C01288=1030.437,28.249,406.907,168.260,43.645,158.132
C01289=1030.444,28.536,406.888,168.262,43.643,158.132
C01290=1030.450,28.786,406.873,168.265,43.641,158.132
C01291=1030.456,29.035,406.856,168.267,43.640,158.131
C01292=1030.462,29.284,406.841,168.269,43.638,158.131
C01293=1030.468,29.533,406.824,168.272,43.637,158.131
C01294=1030.474,29.783,406.808,168.274,43.635,158.131
C01295=1030.480,30.032,406.792,168.277,43.634,158.131
C01296=1030.487,30.281,406.776,168.279,43.632,158.131
C01297=1030.493,30.530,406.760,168.281,43.630,158.131
C01298=1030.499,30.780,406.743,168.284,43.629,158.131
C01299=1030.506,31.030,406.728,168.286,43.627,158.131
C01300=1030.512,31.279,406.712,168.289,43.626,158.131
C01301=1030.518,31.529,406.696,168.291,43.624,158.131
C01302=1030.524,31.778,406.680,168.294,43.623,158.131
C01303=1030.530,32.027,406.664,168.296,43.621,158.130
C01304=1030.537,32.277,406.647,168.298,43.619,158.130
C01305=1030.543,32.527,406.631,168.301,43.618,158.130
C01306=1030.549,32.776,406.615,168.303,43.616,158.130
C01307=1030.555,33.025,406.599,168.305,43.615,158.130
C01308=1030.561,33.274,406.583,168.308,43.613,158.130
C01309=1030.568,33.523,406.567,168.310,43.612,158.130
C01310=1030.575,33.773,406.551,168.312,43.611,158.130
C01311=1030.581,34.023,406.534,168.315,43.609,158.130
C01312=1030.587,34.272,406.519,168.318,43.607,158.130
C01313=1030.593,34.521,406.502,168.319,43.606,158.129
C01314=1030.599,34.770,406.486,168.322,43.604,158.129
C01315=1030.606,35.021,406.470,168.325,43.602,158.129
C01316=1030.612,35.270,406.454,168.326,43.601,158.129
C01317=1030.618,35.519,406.438,168.329,43.599,158.129
C01318=1030.624,35.768,406.421,168.332,43.598,158.129
C01319=1030.631,36.018,406.405,168.333,43.596,158.129
C01320=1030.638,36.267,406.389,168.336,43.594,158.129
C01321=1030.643,36.517,406.373,168.339,43.593,158.129
C01322=1030.650,36.765,406.356,168.341,43.591,158.129
C01323=1030.657,37.015,406.340,168.343,43.590,158.128
C01324=1030.663,37.265,406.324,168.346,43.588,158.128
C01325=1030.669,37.514,406.307,168.348,43.587,158.128
C01326=1030.675,37.763,406.291,168.350,43.585,158.128
C01327=1030.681,38.013,406.274,168.353,43.584,158.128
C01328=1030.687,38.263,406.258,168.355,43.583,158.128
C01329=1030.694,38.511,406.241,168.358,43.581,158.128
C01330=1030.700,38.761,406.225,168.360,43.579,158.128
C01331=1030.706,39.010,406.209,168.362,43.578,158.128
C01332=1030.712,39.260,406.192,168.365,43.576,158.128
C01333=1030.718,39.509,406.176,168.366,43.575,158.128
C01334=1030.724,39.758,406.159,168.369,43.573,158.127
C01335=1030.731,40.008,406.142,168.372,43.572,158.127
C01336=1030.737,40.258,406.126,168.373,43.570,158.127
C01337=1030.743,40.507,406.110,168.376,43.569,158.127
C01338=1030.749,40.756,406.093,168.379,43.567,158.127
C01339=1030.756,41.006,406.076,168.381,43.565,158.127
C01340=1030.761,41.255,406.060,168.383,43.564,158.127
C01341=1030.768,41.504,406.043,168.386,43.562,158.127
C01342=1030.774,41.754,406.026,168.388,43.561,158.127
C01343=1030.781,42.003,406.011,168.390,43.559,158.127
C01344=1030.787,42.252,405.994,168.392,43.558,158.127
C01345=1030.793,42.501,405.977,168.395,43.557,158.127
C01346=1030.800,42.751,405.961,168.398,43.555,158.126
C01347=1030.806,43.000,405.945,168.399,43.554,158.126
C01348=1030.811,43.249,405.927,168.402,43.552,158.126
C01349=1030.818,43.499,405.910,168.405,43.551,158.126
C01350=1030.825,43.785,405.890,168.407,43.549,158.126
C01351=1030.832,44.071,405.872,168.409,43.548,158.126
C01352=1030.838,44.357,405.853,168.412,43.546,158.126
C01353=1030.846,44.643,405.833,168.415,43.544,158.126
C01354=1030.851,44.893,405.817,168.417,43.543,158.126
C01355=1030.858,45.142,405.799,168.420,43.542,158.126
C01356=1030.864,45.392,405.783,168.422,43.540,158.126
C01357=1030.870,45.640,405.766,168.425,43.539,158.126
C01358=1030.876,45.891,405.749,168.426,43.537,158.125
C01359=1030.882,46.139,405.732,168.429,43.536,158.125
C01360=1030.888,46.389,405.716,168.432,43.534,158.125
C01361=1030.895,46.638,405.698,168.434,43.533,158.125
C01362=1030.901,46.887,405.682,168.436,43.531,158.125
C01363=1030.907,47.136,405.664,168.438,43.530,158.125
C01364=1030.913,47.387,405.648,168.441,43.528,158.125
C01365=1030.919,47.635,405.631,168.443,43.527,158.125
C01366=1030.925,47.885,405.615,168.445,43.525,158.125
C01367=1030.931,48.134,405.597,168.448,43.524,158.125
C01368=1030.937,48.384,405.580,168.450,43.522,158.125
C01369=1030.944,48.633,405.563,168.452,43.521,158.125
C01370=1030.950,48.882,405.546,168.454,43.519,158.124
C01371=1030.956,49.132,405.529,168.457,43.518,158.124
C01372=1030.963,49.381,405.512,168.459,43.516,158.124
C01373=1030.968,49.630,405.496,168.461,43.515,158.124
C01374=1030.975,49.880,405.478,168.464,43.514,158.124
C01375=1030.981,50.129,405.461,168.467,43.512,158.124
C01376=1030.987,50.378,405.445,168.468,43.511,158.124
C01377=1030.994,50.628,405.427,168.471,43.509,158.124
C01378=1030.999,50.877,405.410,168.473,43.508,158.124
C01379=1031.006,51.127,405.393,168.476,43.507,158.124
C01380=1031.012,51.375,405.376,168.478,43.505,158.124
C01381=1031.018,51.625,405.360,168.480,43.504,158.124
C01382=1031.024,51.874,405.342,168.483,43.502,158.123
C01383=1031.030,52.123,405.325,168.484,43.501,158.123
C01384=1031.037,52.373,405.308,168.487,43.499,158.123
C01385=1031.043,52.622,405.291,168.490,43.498,158.123
C01386=1031.049,52.872,405.273,168.492,43.496,158.123
C01387=1031.055,53.121,405.257,168.494,43.494,158.123
C01388=1031.062,53.370,405.240,168.496,43.493,158.123
C01389=1031.068,53.619,405.223,168.499,43.491,158.123
C01390=1031.074,53.870,405.206,168.501,43.490,158.123
C01391=1031.080,54.118,405.189,168.503,43.488,158.123
C01392=1031.087,54.368,405.171,168.506,43.487,158.123
C01393=1031.092,54.617,405.154,168.508,43.486,158.122
C01394=1031.099,54.867,405.137,168.510,43.484,158.122
C01395=1031.106,55.116,405.120,168.513,43.483,158.122
C01396=1031.112,55.365,405.103,168.515,43.481,158.122
C01397=1031.118,55.615,405.086,168.517,43.480,158.122
C01398=1031.125,55.864,405.069,168.520,43.478,158.122
C01399=1031.131,56.113,405.052,168.522,43.477,158.122
C01400=1031.137,56.363,405.034,168.525,43.475,158.122
C01401=1031.143,56.612,405.017,168.526,43.473,158.122
C01402=1031.150,56.861,405.000,168.529,43.472,158.122
C01403=1031.156,57.110,404.983,168.532,43.470,158.121
C01404=1031.162,57.360,404.965,168.533,43.469,158.121
C01405=1031.168,57.609,404.948,168.536,43.467,158.121
C01406=1031.175,57.859,404.932,168.539,43.465,158.121
C01407=1031.180,58.108,404.914,168.540,43.464,158.121
C01408=1031.187,58.357,404.897,168.543,43.463,158.121
C01409=1031.194,58.606,404.879,168.545,43.462,158.121
C01410=1031.200,58.856,404.862,168.548,43.460,158.121
C01411=1031.207,59.105,404.844,168.550,43.458,158.121
C01412=1031.212,59.354,404.828,168.552,43.457,158.121
C01413=1031.219,59.604,404.811,168.555,43.455,158.120
C01414=1031.226,59.890,404.791,168.557,43.453,158.120
C01415=1031.234,60.175,404.770,168.560,43.451,158.120
C01416=1031.241,60.461,404.751,168.563,43.449,158.120
C01417=1031.248,60.747,404.731,168.565,43.448,158.120
C01418=1031.254,60.995,404.714,168.568,43.446,158.120
C01419=1031.261,61.245,404.696,168.570,43.445,158.120
C01420=1031.267,61.495,404.679,168.572,43.443,158.120
C01421=1031.273,61.744,404.662,168.575,43.442,158.120
C01422=1031.280,61.993,404.645,168.577,43.440,158.119
C01423=1031.286,62.243,404.627,168.579,43.439,158.119
C01424=1031.293,62.492,404.610,168.582,43.437,158.119
C01425=1031.299,62.741,404.593,168.584,43.435,158.119
C01426=1031.305,62.990,404.575,168.587,43.434,158.119
C01427=1031.312,63.240,404.558,168.589,43.432,158.119
C01428=1031.319,63.489,404.541,168.591,43.430,158.119
C01429=1031.324,63.738,404.523,168.594,43.429,158.119
C01430=1031.330,63.988,404.505,168.595,43.428,158.118
C01431=1031.337,64.237,404.488,168.598,43.426,158.118
C01432=1031.343,64.486,404.470,168.601,43.425,158.118
C01433=1031.350,64.736,404.453,168.603,43.424,158.118
C01434=1031.356,64.985,404.435,168.605,43.422,158.118
C01435=1031.361,65.234,404.417,168.607,43.421,158.118
C01436=1031.368,65.483,404.399,168.610,43.419,158.118
C01437=1031.374,65.732,404.382,168.612,43.418,158.118
C01438=1031.381,65.982,404.364,168.614,43.416,158.118
C01439=1031.387,66.231,404.346,168.617,43.415,158.118
C01440=1031.392,66.481,404.329,168.619,43.413,158.118
C01441=1031.399,66.730,404.312,168.621,43.412,158.118
C01442=1031.405,66.980,404.294,168.623,43.410,158.117
C01443=1031.412,67.228,404.276,168.626,43.409,158.117
C01444=1031.418,67.478,404.258,168.628,43.407,158.117
C01445=1031.424,67.727,404.240,168.630,43.406,158.117
C01446=1031.430,67.976,404.223,168.633,43.404,158.117
C01447=1031.437,68.226,404.205,168.634,43.403,158.117
C01448=1031.443,68.475,404.186,168.637,43.401,158.117
C01449=1031.449,68.724,404.169,168.640,43.400,158.117
C01450=1031.455,68.973,404.152,168.642,43.399,158.117
C01451=1031.462,69.223,404.134,168.644,43.397,158.117
C01452=1031.468,69.473,404.116,168.646,43.396,158.117
C01453=1031.474,69.721,404.098,168.649,43.394,158.117
C01454=1031.480,69.971,404.080,168.652,43.393,158.116
C01455=1031.486,70.220,404.062,168.654,43.392,158.116
C01456=1031.492,70.469,404.044,168.656,43.390,158.116
C01457=1031.498,70.719,404.026,168.658,43.389,158.116
C01458=1031.505,70.968,404.009,168.661,43.387,158.116
C01459=1031.511,71.217,403.991,168.662,43.386,158.116
C01460=1031.517,71.466,403.972,168.665,43.384,158.116
C01461=1031.523,71.716,403.954,168.668,43.383,158.116
C01462=1031.529,71.966,403.937,168.669,43.381,158.116
C01463=1031.535,72.214,403.918,168.672,43.380,158.116
C01464=1031.542,72.464,403.901,168.674,43.378,158.115
C01465=1031.549,72.713,403.882,168.677,43.377,158.115
C01466=1031.554,72.962,403.865,168.678,43.375,158.115
C01467=1031.560,73.211,403.847,168.681,43.374,158.115
C01468=1031.567,73.461,403.828,168.684,43.372,158.115
C01469=1031.573,73.710,403.810,168.686,43.371,158.115
C01470=1031.579,73.959,403.793,168.688,43.370,158.115
C01471=1031.585,74.208,403.775,168.690,43.369,158.115
C01472=1031.592,74.458,403.757,168.693,43.367,158.115
C01473=1031.598,74.707,403.738,168.696,43.366,158.115
C01474=1031.604,74.957,403.720,168.697,43.364,158.115
C01475=1031.610,75.205,403.702,168.700,43.363,158.115
C01476=1031.617,75.455,403.684,168.702,43.361,158.114
C01477=1031.623,75.704,403.666,168.704,43.360,158.114
C01478=1031.630,75.990,403.646,168.707,43.358,158.114
C01479=1031.637,76.275,403.625,168.710,43.356,158.114
C01480=1031.644,76.561,403.604,168.713,43.355,158.114
C01481=1031.651,76.846,403.583,168.715,43.353,158.114
C01482=1031.657,77.096,403.565,168.717,43.351,158.114
C01483=1031.664,77.345,403.547,168.720,43.350,158.114
C01484=1031.670,77.594,403.529,168.722,43.349,158.114
C01485=1031.676,77.844,403.510,168.724,43.347,158.114
C01486=1031.682,78.092,403.492,168.727,43.346,158.114
C01487=1031.688,78.342,403.474,168.729,43.344,158.113
C01488=1031.695,78.591,403.455,168.731,43.343,158.113
C01489=1031.701,78.841,403.437,168.733,43.342,158.113
C01490=1031.707,79.090,403.419,168.736,43.340,158.113
C01491=1031.712,79.338,403.400,168.738,43.339,158.113
C01492=1031.718,79.588,403.382,168.740,43.338,158.113
C01493=1031.725,79.837,403.363,168.743,43.336,158.113
C01494=1031.731,80.086,403.344,168.745,43.335,158.113
C01495=1031.737,80.336,403.327,168.748,43.334,158.113
C01496=1031.744,80.585,403.308,168.749,43.333,158.113
C01497=1031.750,80.834,403.290,168.752,43.331,158.113
C01498=1031.756,81.083,403.272,168.754,43.330,158.113
C01499=1031.761,81.333,403.252,168.756,43.328,158.112
C01500=1031.768,81.582,403.234,168.759,43.327,158.112
C01501=1031.774,81.832,403.216,168.761,43.326,158.112
C01502=1031.780,82.081,403.197,168.764,43.324,158.112
C01503=1031.786,82.329,403.179,168.766,43.323,158.112
C01504=1031.792,82.579,403.161,168.768,43.321,158.112
C01505=1031.799,82.828,403.142,168.770,43.320,158.112
C01506=1031.805,83.077,403.124,168.773,43.318,158.112
C01507=1031.811,83.327,403.104,168.776,43.317,158.112
C01508=1031.817,83.576,403.087,168.777,43.316,158.112
C01509=1031.823,83.826,403.068,168.780,43.314,158.112
C01510=1031.830,84.075,403.049,168.782,43.313,158.112
C01511=1031.836,84.323,403.031,168.784,43.311,158.111
C01512=1031.842,84.573,403.013,168.787,43.310,158.111
C01513=1031.848,84.822,402.994,168.789,43.308,158.111
C01514=1031.855,85.071,402.976,168.792,43.307,158.111
C01515=1031.860,85.321,402.956,168.793,43.306,158.111
C01516=1031.867,85.570,402.938,168.796,43.304,158.111
C01517=1031.873,85.819,402.920,168.798,43.303,158.111
C01518=1031.879,86.069,402.901,168.801,43.301,158.111
C01519=1031.886,86.318,402.883,168.803,43.300,158.111
C01520=1031.892,86.567,402.864,168.805,43.299,158.111
C01521=1031.899,86.816,402.845,168.808,43.297,158.111
C01522=1031.904,87.066,402.827,168.810,43.296,158.110
C01523=1031.910,87.315,402.808,168.812,43.295,158.110
C01524=1031.916,87.563,402.790,168.815,43.293,158.110
C01525=1031.923,87.813,402.771,168.817,43.292,158.110
C01526=1031.929,88.062,402.753,168.819,43.290,158.110
C01527=1031.936,88.311,402.734,168.821,43.289,158.110
C01528=1031.941,88.560,402.715,168.824,43.287,158.110
C01529=1031.948,88.809,402.696,168.827,43.286,158.110
C01530=1031.954,89.059,402.678,168.828,43.284,158.110
C01531=1031.960,89.308,402.659,168.831,43.283,158.110
C01532=1031.967,89.557,402.641,168.834,43.281,158.110
C01533=1031.973,89.807,402.622,168.836,43.280,158.110
C01534=1031.979,90.056,402.603,168.838,43.278,158.109
C01535=1031.985,90.305,402.584,168.840,43.277,158.109
C01536=1031.991,90.555,402.565,168.843,43.276,158.109
C01537=1031.997,90.804,402.546,168.845,43.275,158.109
C01538=1032.003,91.053,402.527,168.847,43.273,158.109
C01539=1032.009,91.302,402.508,168.850,43.272,158.109
C01540=1032.016,91.551,402.490,168.852,43.270,158.109
C01541=1032.022,91.801,402.471,168.855,43.269,158.109
C01542=1032.028,92.086,402.449,168.857,43.267,158.109
C01543=1032.036,92.371,402.426,168.860,43.266,158.109
C01544=1032.042,92.657,402.405,168.862,43.265,158.109
C01545=1032.050,92.942,402.384,168.865,43.263,158.109
C01546=1032.056,93.191,402.364,168.867,43.262,158.108
C01547=1032.062,93.440,402.346,168.870,43.260,158.108
C01548=1032.068,93.690,402.326,168.872,43.259,158.108
C01549=1032.074,93.939,402.308,168.874,43.258,158.108
C01550=1032.080,94.188,402.289,168.876,43.257,158.108
C01551=1032.087,94.438,402.270,168.879,43.255,158.108
C01552=1032.093,94.688,402.250,168.882,43.254,158.108
C01553=1032.099,94.936,402.231,168.884,43.253,158.108
C01554=1032.106,95.185,402.212,168.886,43.251,158.108
C01555=1032.111,95.435,402.193,168.888,43.250,158.108
C01556=1032.118,95.684,402.174,168.891,43.248,158.108
C01557=1032.123,95.933,402.155,168.894,43.247,158.108
C01558=1032.130,96.182,402.137,168.895,43.246,158.108
C01559=1032.136,96.431,402.117,168.898,43.244,158.107
C01560=1032.142,96.680,402.098,168.900,43.243,158.107
C01561=1032.148,96.930,402.079,168.902,43.241,158.107
C01562=1032.154,97.179,402.060,168.905,43.240,158.107
C01563=1032.160,97.428,402.041,168.907,43.239,158.107
C01564=1032.167,97.677,402.021,168.910,43.237,158.107
C01565=1032.173,97.926,402.002,168.912,43.236,158.107
C01566=1032.179,98.175,401.984,168.914,43.234,158.107
C01567=1032.185,98.425,401.964,168.917,43.233,158.107
C01568=1032.192,98.674,401.945,168.919,43.232,158.107
C01569=1032.198,98.923,401.926,168.921,43.230,158.107
C01570=1032.204,99.172,401.907,168.923,43.229,158.107
C01571=1032.211,99.422,401.888,168.926,43.227,158.106
C01572=1032.217,99.670,401.868,168.929,43.226,158.106
C01573=1032.223,99.919,401.849,168.930,43.224,158.106
C01574=1032.229,100.169,401.830,168.933,43.223,158.106
C01575=1032.235,100.418,401.810,168.935,43.222,158.106
C01576=1032.241,100.668,401.791,168.938,43.220,158.106
C01577=1032.247,100.917,401.772,168.940,43.219,158.106
C01578=1032.253,101.166,401.752,168.942,43.218,158.106
C01579=1032.259,101.415,401.733,168.945,43.217,158.106
C01580=1032.266,101.664,401.713,168.947,43.215,158.106
C01581=1032.271,101.913,401.694,168.950,43.214,158.106
C01582=1032.277,102.163,401.675,168.951,43.213,158.106
C01583=1032.283,102.411,401.655,168.954,43.211,158.106
C01584=1032.290,102.661,401.636,168.957,43.210,158.106
C01585=1032.296,102.910,401.616,168.959,43.209,158.106
C01586=1032.302,103.160,401.597,168.961,43.207,158.105
C01587=1032.308,103.408,401.577,168.963,43.206,158.105
C01588=1032.314,103.657,401.558,168.966,43.205,158.105
C01589=1032.320,103.906,401.538,168.969,43.204,158.105
C01590=1032.326,104.156,401.519,168.970,43.202,158.105
C01591=1032.333,104.405,401.499,168.973,43.201,158.105
C01592=1032.339,104.654,401.480,168.975,43.200,158.105
C01593=1032.345,104.903,401.460,168.978,43.198,158.105
C01594=1032.351,105.153,401.441,168.981,43.197,158.105
C01595=1032.357,105.401,401.421,168.982,43.196,158.105
C01596=1032.362,105.651,401.402,168.985,43.194,158.105
C01597=1032.370,105.900,401.382,168.987,43.193,158.105
C01598=1032.375,106.149,401.363,168.990,43.192,158.105
C01599=1032.381,106.398,401.343,168.992,43.190,158.104
C01600=1032.387,106.648,401.323,168.994,43.189,158.104
C01601=1032.394,106.896,401.304,168.997,43.188,158.104
C01602=1032.400,107.146,401.284,169.000,43.186,158.104
C01603=1032.406,107.395,401.264,169.001,43.185,158.104
C01604=1032.412,107.644,401.244,169.004,43.184,158.104
C01605=1032.418,107.893,401.226,169.006,43.183,158.104
C01606=1032.425,108.179,401.203,169.009,43.181,158.104
C01607=1032.433,108.464,401.180,169.011,43.180,158.104
C01608=1032.440,108.749,401.158,169.015,43.178,158.104
C01609=1032.447,109.035,401.135,169.018,43.176,158.104
C01610=1032.453,109.284,401.116,169.020,43.175,158.104
C01611=1032.459,109.533,401.096,169.022,43.174,158.104
C01612=1032.465,109.783,401.076,169.024,43.173,158.103
C01613=1032.471,110.031,401.056,169.027,43.171,158.103
C01614=1032.478,110.281,401.037,169.030,43.170,158.103
C01615=1032.484,110.530,401.017,169.031,43.169,158.103
C01616=1032.490,110.779,400.997,169.034,43.167,158.103
C01617=1032.496,111.028,400.978,169.037,43.166,158.103
C01618=1032.502,111.277,400.958,169.039,43.165,158.103
C01619=1032.509,111.527,400.938,169.042,43.163,158.103
C01620=1032.515,111.775,400.918,169.043,43.162,158.103
C01621=1032.520,112.025,400.898,169.046,43.161,158.103
C01622=1032.526,112.274,400.878,169.049,43.159,158.103
C01623=1032.533,112.523,400.858,169.051,43.158,158.103
C01624=1032.539,112.772,400.838,169.053,43.157,158.103
C01625=1032.545,113.021,400.819,169.056,43.155,158.103
C01626=1032.551,113.271,400.799,169.058,43.154,158.103
C01627=1032.557,113.520,400.779,169.061,43.153,158.103
C01628=1032.563,113.769,400.759,169.063,43.152,158.103
C01629=1032.569,114.018,400.738,169.065,43.150,158.102
C01630=1032.575,114.267,400.718,169.068,43.149,158.102
C01631=1032.581,114.516,400.698,169.070,43.148,158.102
C01632=1032.587,114.765,400.678,169.073,43.147,158.102
C01633=1032.593,115.014,400.658,169.075,43.146,158.102
C01634=1032.599,115.264,400.638,169.077,43.145,158.102
C01635=1032.605,115.513,400.618,169.080,43.143,158.102
C01636=1032.611,115.762,400.598,169.082,43.142,158.102
C01637=1032.617,116.011,400.577,169.085,43.141,158.102
C01638=1032.623,116.260,400.557,169.087,43.140,158.102
C01639=1032.629,116.509,400.537,169.089,43.139,158.102
C01640=1032.635,116.759,400.517,169.092,43.138,158.102
C01641=1032.641,117.008,400.497,169.094,43.136,158.102
C01642=1032.647,117.256,400.477,169.097,43.135,158.102
C01643=1032.652,117.505,400.456,169.098,43.134,158.102
C01644=1032.659,117.755,400.436,169.101,43.133,158.102
C01645=1032.665,118.004,400.416,169.104,43.131,158.102
C01646=1032.671,118.253,400.396,169.106,43.130,158.102
C01647=1032.677,118.502,400.375,169.109,43.129,158.101
C01648=1032.683,118.751,400.355,169.111,43.128,158.101
C01649=1032.689,119.001,400.335,169.113,43.127,158.101
C01650=1032.695,119.250,400.315,169.116,43.125,158.101
C01651=1032.701,119.498,400.293,169.119,43.124,158.101
C01652=1032.708,119.748,400.273,169.121,43.123,158.101
C01653=1032.714,119.996,400.253,169.123,43.121,158.101
C01654=1032.720,120.245,400.233,169.125,43.120,158.101
C01655=1032.725,120.495,400.212,169.128,43.119,158.101
C01656=1032.731,120.744,400.192,169.131,43.118,158.101
C01657=1032.737,120.993,400.172,169.133,43.117,158.101
C01658=1032.744,121.242,400.152,169.135,43.115,158.101
C01659=1032.749,121.491,400.131,169.138,43.114,158.101
C01660=1032.756,121.741,400.111,169.140,43.113,158.101
C01661=1032.762,121.989,400.090,169.143,43.112,158.101
C01662=1032.769,122.239,400.070,169.146,43.111,158.101
C01663=1032.774,122.488,400.050,169.147,43.109,158.101
C01664=1032.780,122.736,400.030,169.150,43.108,158.101
C01665=1032.787,122.986,400.009,169.153,43.107,158.101
C01666=1032.793,123.235,399.989,169.155,43.106,158.101
C01667=1032.799,123.484,399.968,169.157,43.104,158.100
C01668=1032.805,123.733,399.948,169.160,43.103,158.100
C01669=1032.811,123.982,399.927,169.162,43.102,158.100
C01670=1032.818,124.267,399.904,169.165,43.101,158.100
C01671=1032.825,124.552,399.880,169.169,43.099,158.100
C01672=1032.832,124.837,399.857,169.171,43.097,158.100
C01673=1032.839,125.123,399.834,169.174,43.096,158.100
C01674=1032.845,125.372,399.813,169.176,43.095,158.100
C01675=1032.851,125.622,399.793,169.179,43.093,158.100
C01676=1032.857,125.870,399.773,169.182,43.092,158.100
C01677=1032.864,126.120,399.753,169.183,43.091,158.100
C01678=1032.869,126.368,399.731,169.186,43.089,158.100
C01679=1032.876,126.618,399.711,169.189,43.088,158.100
C01680=1032.882,126.867,399.691,169.192,43.087,158.100
C01681=1032.889,127.116,399.670,169.194,43.086,158.100
C01682=1032.894,127.365,399.649,169.196,43.084,158.100
C01683=1032.901,127.614,399.629,169.199,43.083,158.100
C01684=1032.907,127.864,399.609,169.201,43.082,158.099
C01685=1032.913,128.112,399.588,169.204,43.081,158.099
C01686=1032.920,128.362,399.567,169.206,43.079,158.099
C01687=1032.926,128.611,399.547,169.209,43.078,158.099
C01688=1032.932,128.859,399.526,169.211,43.077,158.099
C01689=1032.938,129.109,399.506,169.214,43.076,158.099
C01690=1032.945,129.357,399.485,169.216,43.074,158.099
C01691=1032.951,129.606,399.465,169.218,43.073,158.099
C01692=1032.956,129.856,399.444,169.221,43.072,158.099
C01693=1032.963,130.104,399.423,169.224,43.071,158.099
C01694=1032.969,130.354,399.403,169.227,43.069,158.099
C01695=1032.976,130.603,399.382,169.228,43.068,158.099
C01696=1032.982,130.852,399.361,169.231,43.067,158.099
C01697=1032.987,131.102,399.340,169.234,43.066,158.099
C01698=1032.994,131.350,399.320,169.236,43.065,158.099
C01699=1033.000,131.600,399.299,169.239,43.063,158.099
C01700=1033.006,131.848,399.278,169.242,43.062,158.099
C01701=1033.012,132.098,399.257,169.244,43.061,158.099
C01702=1033.018,132.347,399.235,169.246,43.060,158.099
C01703=1033.024,132.595,399.215,169.249,43.059,158.099
C01704=1033.030,132.845,399.194,169.252,43.057,158.098
C01705=1033.036,133.093,399.173,169.253,43.056,158.098
C01706=1033.042,133.343,399.152,169.256,43.055,158.098
C01707=1033.048,133.591,399.131,169.259,43.054,158.098
C01708=1033.054,133.841,399.111,169.261,43.053,158.098
C01709=1033.060,134.090,399.089,169.264,43.052,158.098
C01710=1033.067,134.338,399.068,169.267,43.051,158.098
C01711=1033.073,134.588,399.047,169.270,43.049,158.098
C01712=1033.078,134.837,399.026,169.271,43.048,158.098
C01713=1033.085,135.086,399.005,169.274,43.047,158.098
C01714=1033.091,135.335,398.984,169.277,43.046,158.098
C01715=1033.097,135.584,398.963,169.280,43.044,158.098
C01716=1033.103,135.833,398.943,169.281,43.043,158.098
C01717=1033.109,136.082,398.921,169.284,43.042,158.098
C01718=1033.116,136.331,398.900,169.287,43.041,158.098
C01719=1033.121,136.581,398.879,169.289,43.040,158.098
C01720=1033.127,136.829,398.858,169.292,43.039,158.098
C01721=1033.134,137.078,398.837,169.295,43.038,158.098
C01722=1033.140,137.327,398.815,169.297,43.036,158.098
C01723=1033.145,137.576,398.795,169.299,43.035,158.098
C01724=1033.151,137.826,398.773,169.302,43.034,158.098
C01725=1033.158,138.074,398.752,169.305,43.033,158.098
C01726=1033.164,138.323,398.731,169.308,43.032,158.098
C01727=1033.170,138.573,398.710,169.310,43.031,158.098
C01728=1033.177,138.822,398.689,169.312,43.030,158.098
C01729=1033.182,139.070,398.668,169.315,43.029,158.098
C01730=1033.188,139.319,398.646,169.318,43.028,158.098
C01731=1033.194,139.568,398.625,169.320,43.027,158.098
C01732=1033.200,139.818,398.604,169.323,43.025,158.098
C01733=1033.206,140.067,398.582,169.326,43.024,158.098
C01734=1033.213,140.352,398.558,169.328,43.022,158.097
C01735=1033.220,140.637,398.533,169.331,43.021,158.097
C01736=1033.227,140.922,398.509,169.334,43.020,158.097
C01737=1033.233,141.207,398.484,169.337,43.019,158.097
C01738=1033.240,141.456,398.463,169.340,43.018,158.097
C01739=1033.246,141.705,398.442,169.342,43.017,158.097
C01740=1033.252,141.954,398.420,169.345,43.015,158.097
C01741=1033.258,142.203,398.399,169.347,43.015,158.097
C01742=1033.264,142.428,398.380,169.350,43.013,158.097
C01743=1033.269,142.653,398.360,169.352,43.012,158.097
C01744=1033.275,142.878,398.341,169.355,43.012,158.097
C01745=1033.280,143.102,398.321,169.357,43.011,158.097
C01746=1033.286,143.327,398.302,169.359,43.010,158.097
C01747=1033.291,143.552,398.282,169.361,43.009,158.097
C01748=1033.296,143.776,398.264,169.364,43.008,158.097
C01749=1033.302,144.001,398.243,169.366,43.007,158.097
C01750=1033.309,144.250,398.222,169.369,43.005,158.097
C01751=1033.314,144.499,398.201,169.372,43.004,158.097
C01752=1033.320,144.748,398.179,169.374,43.003,158.097
C01753=1033.327,144.997,398.158,169.376,43.002,158.097
C01754=1033.333,145.246,398.136,169.379,43.001,158.097
C01755=1033.338,145.495,398.115,169.382,43.000,158.097
C01756=1033.344,145.744,398.093,169.385,42.999,158.097
C01757=1033.351,145.993,398.072,169.388,42.997,158.097
C01758=1033.357,146.243,398.050,169.389,42.996,158.097
C01759=1033.364,146.491,398.029,169.392,42.995,158.097
C01760=1033.369,146.740,398.008,169.395,42.994,158.097
C01761=1033.375,146.990,397.985,169.398,42.993,158.097
C01762=1033.381,147.239,397.964,169.400,42.992,158.097
C01763=1033.387,147.488,397.942,169.403,42.991,158.097
C01764=1033.393,147.737,397.921,169.406,42.990,158.097
C01765=1033.399,147.985,397.899,169.409,42.989,158.097
C01766=1033.405,148.234,397.877,169.411,42.988,158.097
C01767=1033.411,148.483,397.855,169.413,42.987,158.097
C01768=1033.418,148.733,397.834,169.416,42.986,158.097
C01769=1033.424,148.982,397.812,169.419,42.985,158.097
C01770=1033.430,149.230,397.790,169.422,42.984,158.097
C01771=1033.436,149.479,397.768,169.425,42.982,158.097
C01772=1033.442,149.728,397.747,169.426,42.981,158.097
C01773=1033.447,149.978,397.725,169.429,42.981,158.097
C01774=1033.454,150.226,397.702,169.432,42.980,158.097
C01775=1033.459,150.475,397.681,169.435,42.979,158.097
C01776=1033.465,150.724,397.659,169.438,42.978,158.097
C01777=1033.472,150.973,397.638,169.440,42.977,158.097
C01778=1033.478,151.222,397.615,169.443,42.975,158.097
C01779=1033.484,151.471,397.593,169.445,42.974,158.097
C01780=1033.490,151.720,397.571,169.448,42.974,158.097
C01781=1033.496,151.969,397.549,169.451,42.973,158.097
C01782=1033.502,152.218,397.528,169.453,42.972,158.097
C01783=1033.508,152.467,397.506,169.456,42.970,158.097
C01784=1033.514,152.715,397.484,169.459,42.969,158.097
C01785=1033.520,152.965,397.462,169.462,42.968,158.097
C01786=1033.526,153.214,397.440,169.464,42.967,158.097
C01787=1033.532,153.463,397.418,169.468,42.966,158.097
C01788=1033.539,153.712,397.396,169.469,42.965,158.097
C01789=1033.545,153.961,397.374,169.472,42.964,158.097
C01790=1033.550,154.210,397.351,169.475,42.963,158.097
C01791=1033.557,154.459,397.330,169.478,42.962,158.097
C01792=1033.563,154.707,397.308,169.481,42.961,158.097
C01793=1033.569,154.956,397.286,169.484,42.960,158.097
C01794=1033.574,155.205,397.263,169.486,42.959,158.097
C01795=1033.581,155.454,397.242,169.488,42.958,158.097
C01796=1033.587,155.703,397.219,169.491,42.957,158.097
C01797=1033.592,155.952,397.197,169.494,42.956,158.097
C01798=1033.601,156.286,397.167,169.498,42.955,158.097
C01799=1033.609,156.619,397.138,169.502,42.953,158.097
C01800=1033.617,156.952,397.108,169.505,42.952,158.097
C01801=1033.626,157.285,397.078,169.508,42.951,158.097
C01802=1033.631,157.535,397.056,169.511,42.950,158.097
C01803=1033.638,157.783,397.034,169.514,42.949,158.097
C01804=1033.644,158.032,397.012,169.517,42.948,158.097
C01805=1033.649,158.281,396.989,169.520,42.947,158.097
C01806=1033.656,158.531,396.967,169.523,42.946,158.097
C01807=1033.662,158.779,396.945,169.525,42.945,158.097
C01808=1033.668,159.028,396.922,169.528,42.944,158.097
C01809=1033.674,159.277,396.900,169.531,42.943,158.097
C01810=1033.680,159.526,396.878,169.533,42.942,158.097
C01811=1033.686,159.775,396.855,169.536,42.941,158.097
C01812=1033.692,160.024,396.833,169.539,42.940,158.097
C01813=1033.698,160.273,396.810,169.542,42.939,158.097
C01814=1033.703,160.521,396.788,169.544,42.939,158.097
C01815=1033.709,160.770,396.765,169.547,42.938,158.097
C01816=1033.715,161.019,396.743,169.550,42.937,158.097
C01817=1033.721,161.268,396.720,169.553,42.936,158.097
